METHOD PRIVATE ReferenceHMI
VAR_INPUT
END_VAR
Service_Handshake.AllocateMoveStructure 				REF= GVL_ADS.AllocateMoveStructure;
Service_Handshake.AllocateMoveStructure_Reverse 		REF= GVL_ADS.AllocateMoveStructure_Reverse;
Service_Handshake.EmptyRobotToTurnTableMove 			REF= GVL_ADS.EmptyRobotToTurnTableMove;
Service_Handshake.AllocateCircleMove 					REF= GVL_ADS.AllocateCircleMove;
Service_Handshake.TurnTableMove 						REF= GVL_ADS.TurnTableMove;
//Service_Handshake.AxesControl REF= GVL_ADS.AxesControl;
Service_Handshake.MachineReset 							REF= GVL_ADS.MachineReset;
Service_Handshake.RareFullBoxPush 						REF= GVL_ADS.RareFullBoxPush;
Service_Handshake.AutoMode_AllocateCircleMove 			REF= GVL_ADS.AutoMode_AllocateCircleMove;
Service_Handshake.AutoMode_RobotWarehouseMove 			REF= GVL_ADS.AutoMode_RobotWarehouseMove;
Service_Handshake.AutoMode_RobotAbsMove 				REF= GVL_ADS.AutoMode_RobotAbsMove;
Service_Handshake.AutoMode_EmptyBoxMove 				REF= GVL_ADS.AutoMode_EmptyBoxMove;
Service_Handshake.AutoMode_TurnTableMOve 				REF= GVL_ADS.AutoMode_TurnTableMOve;
Service_Handshake.AutoMode_AllocateMove 				REF= GVL_ADS.AutoMode_AllocateMove;
Service_Handshake.AutoMode_AllocateMove_Reverse 		REF= GVL_ADS.AutoMode_AllocateMove_Reverse;
Service_Handshake.AutoMode_AllocateBatchMode 			REF= GVL_ADS.AutoMode_AllocateBatchMode;
Service_Handshake.AutoMode_AllocateBatchMode_Reverse 	REF= GVL_ADS.AutoMode_AllocateBatchMode_Reverse;
Service_Handshake.AutoMode_SimpleAllocation_Batch 		REF= GVL_ADS.AutoMode_SimpleAllocation_Batch;
Service_Handshake.AutoMode_RareBoxMove 					REF= GVL_ADS.AutoMode_RareBoxMove;
Service_Handshake.AutoMode_OutBoxMove 					REF= GVL_ADS.AutoMode_OutBoxMove;
Service_Handshake.AutoMode_BoxMoveReverse 				REF= GVL_ADS.AutoMode_BoxMoveReverse;
Service_Handshake.AutoMode_WarehouseMove 				REF= GVL_ADS.AutoMode_WarehouseMove;
Service_Handshake.AutoMode_ErrorHandle 					REF= GVL_ADS.AutoMode_ErrorHandle;
Service_Handshake.AlarmAllocation 						REF= GVL_ADS.AlarmAllocation;
Service_Handshake.AutoMode_MoveConveyorJob 				REF= GVL_ADS.AutoMode_MoveConveyorJob;
Service_Handshake.AutoMode_WarehouseMotoWithRobotMove 	REF= GVL_ADS.AutoMode_WarehouseMotoWithRobotMove;
Service_Handshake.AutoMode_SimpleAllocate 				REF= GVL_ADS.AutoMode_SimpleAllocate;
Service_Handshake.AutoMode_PullOutConveyor 				REF= GVL_ADS.AutoMode_PullOutConveyor;
Service_Handshake.AutoMode_AddBoxes 					REF= GVL_ADS.AutoMode_AddBoxes;
Service_Handshake.MachineHome 							REF= GVL_ADS.MachineHome;
Service_Handshake.StorageRegionHome 					REF= GVL_ADS.StorageRegionHome;
Service_Handshake.AllocationRegionHome 					REF= GVL_ADS.AllocationRegionHome;
Service_Handshake.FGARegionHome 						REF= GVL_ADS.FGARegionHome;
Service_Handshake.StorageRegionMode 					REF= GVL_ADS.StorageRegionMode;
Service_Handshake.AllocationRegion 						REF= GVL_ADS.AllocationRegion;
Service_Handshake.FGARegionMode 						REF= GVL_ADS.FGARegionMode;
Service_Handshake.MachineMode 							REF= GVL_ADS.MachineMode;
Service_Handshake.OpPannel_Status 						REF= GVL_ADS.OpPannel_Status;
Service_Handshake.OpPannel_Ctrl 						REF= GVL_ADS.OpPannel_Ctrl;
Service_Handshake.FanucRobot_General 					REF= GVL_ADS.FanucRobot_General;
Service_Handshake.AutoMode_FeedInEmptyBoxWithRobot 		REF= GVL_ADS.AutoMode_FeedInEmptyBoxWithRobot;
Service_Handshake.AutoMode_ReloadRoundBeltBoxWithRobot 	REF= GVL_ADS.AutoMode_ReloadRoundBeltBoxWithRobot;
Service_Handshake.AutoMode_UpperFeedInConveyor 			REF= GVL_ADS.AutoMode_UpperFeedInConveyor;
//Service_Handshake.MachineState REF= GVL_ADS.MachineState;
Service_Handshake.AutoMode_RobotRegionMove_FeedInConveyor REF= GVL_ADS.AutoMode_RobotRegionMove_FeedInConveyor;
Service_Handshake.AutoMode_RobotRegionMove_AllocatedConveyor REF= GVL_ADS.AutoMode_RobotRegionMove_AllocatedConveyor;
Service_Handshake.AutoMode_RobotRegionMove_PullOutConveyor REF= GVL_ADS.AutoMode_RobotRegionMove_PullOutConveyor;
Service_Handshake.AutoMode_RobotRegionMove_BufferArea 	REF= GVL_ADS.AutoMode_RobotRegionMove_BufferArea;
Service_Handshake.AutoMode_RobotRegionMove_RoundBelt 	REF= GVL_ADS.AutoMode_RobotRegionMove_RoundBelt;
Service_Handshake.AutoMode_ShippingRobot_Left 			REF= GVL_ADS.AutoMode_ShippingRobot_Left;
Service_Handshake.AutoMode_ShippingRobot_Right 			REF= GVL_ADS.AutoMode_ShippingRobot_Right;
Service_Handshake.AutoMode_ShippingRobot_TransmitCVEnd 	REF= GVL_ADS.AutoMode_ShippingRobot_TransmitCVEnd;
Service_Handshake.AutoMode_SameSizeCVCamera 			REF= GVL_ADS.AutoMode_SameSizeCVCamera;
Service_Handshake.AutoMode_SameSizeCVCamera_Reverse 	REF= GVL_ADS.AutoMode_SameSizeCVCamera_Reverse;
Service_Handshake.AutoMode_DifferentCVCamera 			REF= GVL_ADS.AutoMode_DifferentCVCamera;

Service_Handshake.AllocationRobotNeedlingMove 			REF= GVL_ADS.AllocationRobotNeedlingMove;
Service_Handshake.RebootModbusDevices 					REF= GVL_ADS.RebootModbusDevices;
Service_Handshake.AutoMode_ShippingLeftSideTransCV 		REF= GVL_ADS.AutoMode_ShippingLeftSideTransCV;
Service_Handshake.AutoMode_ShippingRightSideTransCV 	REF= GVL_ADS.AutoMode_ShippingRightSideTransCV;
Service_Handshake.AutoMode_ShippingRobot_Buffer REF= GVL_ADS.AutoMode_ShippingRobot_Buffer;
Service_Handshake.AutoMode_ShippingRobot_PhotoStandByPos REF= GVL_ADS.AutoMode_ShippingRobot_PhotoStandByPos;
Service_Handshake.AutoMode_ShippingRobotTransfer REF= GVL_ADS.AutoMode_ShippingRobotTransfer;
Service_Handshake.AutoMode_ShippingPlateScan REF= GVL_ADS.AutoMode_ShippingPlateScan;

Service_Handshake.AutoMode_FeedInRoundBeltBoxToWareHouse REF= GVL_ADS.AutoMode_FeedInRoundBeltBoxToWareHouse;
Service_Handshake.AutoMode_WareHouseInnerPickToRoundBelt REF= GVL_ADS.AutoMode_WareHouseInnerPickToRoundBelt;
Service_Handshake.AutoMode_WareHouseInnerPickToRoundBeltBatch REF= GVL_ADS.AutoMode_WareHouseInnerPickToRoundBeltBatch;
Service_Handshake.AutoMode_FeedInRoundBeltBoxBatch REF= GVL_ADS.AutoMode_FeedInRoundBeltBoxBatch;

Service_Handshake.AutoMode_RobotSelfHoming REF= GVL_ADS.AutoMode_RobotSelfHoming;

Service_Handshake.AutoMode_ReverseBatchPick REF= GVL_ADS.AutoMode_ReverseBatchPick;
Service_Handshake.AutoMode_ReverseBoxToWareHouse REF= GVL_ADS.AutoMode_ReverseBoxToWareHouse;

Service_Handshake.BuzzCtrl REF= GVL_ADS.BuzzCtrl;
END_METHOD

METHOD RefShippingService
VAR_INPUT
END_VAR
ShippingService.AutoMode_ShippingRobot_Left 			REF= Service_Handshake.AutoMode_ShippingRobot_Left;
ShippingService.AutoMode_ShippingRobot_Right 			REF= Service_Handshake.AutoMode_ShippingRobot_Right;
ShippingService.AutoMode_ShippingRobot_TransmitCVEnd 	REF= Service_Handshake.AutoMode_ShippingRobot_TransmitCVEnd;
ShippingService.AutoMode_ShippingTransCV_LeftSide 		REF= Service_Handshake.AutoMode_ShippingLeftSideTransCV;
ShippingService.AutoMode_ShippingTransCV_RightSide 		REF= Service_Handshake.AutoMode_ShippingRightSideTransCV;
ShippingService.AutoMode_ShippingRobot_Buffer			REF= Service_Handshake.AutoMode_ShippingRobot_Buffer;
ShippingService.AutoMode_ShippingRobot_PhotoStandByPos  REF= Service_Handshake.AutoMode_ShippingRobot_PhotoStandByPos;
ShippingService.AutoMode_ShippingRobotTransfer			REF= Service_Handshake.AutoMode_ShippingRobotTransfer;
ShippingService.AutoMode_ShippingPlateScan				REF= Service_Handshake.AutoMode_ShippingPlateScan;
END_METHOD

METHOD PRIVATE RefStorageService
VAR_INPUT
END_VAR
StorageService.AutoMode_ReloadRoundBeltBoxWithRobot	REF= Service_Handshake.AutoMode_ReloadRoundBeltBoxWithRobot;
StorageService.AutoMode_FeedInEmptyBoxWithRobot REF= Service_Handshake.AutoMode_FeedInEmptyBoxWithRobot;
StorageService.AutoMode_RobotRegionMove_FeedInConveyor REF= Service_Handshake.AutoMode_RobotRegionMove_FeedInConveyor;
StorageService.AutoMode_RobotRegionMove_AllocatedConveyor REF= Service_Handshake.AutoMode_RobotRegionMove_AllocatedConveyor;
StorageService.AutoMode_RobotRegionMove_PullOutConveyor REF= Service_Handshake.AutoMode_RobotRegionMove_PullOutConveyor;
StorageService.AutoMode_RobotRegionMove_BufferArea REF= Service_Handshake.AutoMode_RobotRegionMove_BufferArea;
StorageService.AutoMode_RobotRegionMove_RoundBelt REF= Service_Handshake.AutoMode_RobotRegionMove_RoundBelt;
StorageService.AutoMode_UpperFeedInConveyor REF=  Service_Handshake.AutoMode_UpperFeedInConveyor;
StorageService.AutoMode_AddBoxes REF= Service_Handshake.AutoMode_AddBoxes;
StorageService.AutoMode_PullOutConveyor REF= Service_Handshake.AutoMode_PullOutConveyor;
StorageService.AutoMode_RobotAbsMove REF=  Service_Handshake.AutoMode_RobotAbsMove;
StorageService.AutoMode_WarehouseMotoWithRobotMove REF= Service_Handshake.AutoMode_WarehouseMotoWithRobotMove;
StorageService.RebootModbusDevices REF= Service_Handshake.RebootModbusDevices;
StorageService.AutoMode_FeedInRoundBeltBoxToWareHouse REF= Service_Handshake.AutoMode_FeedInRoundBeltBoxToWareHouse;
StorageService.AutoMode_WareHouseInnerPickToRoundBelt REF= Service_Handshake.AutoMode_WareHouseInnerPickToRoundBelt;
StorageService.AutoMode_WareHouseInnerPickToRoundBeltBatch REF= Service_Handshake.AutoMode_WareHouseInnerPickToRoundBeltBatch;
StorageService.AutoMode_FeedInRoundBeltBoxBatch REF= Service_Handshake.AutoMode_FeedInRoundBeltBoxBatch;
StorageService.AutoMode_RobotSelfHoming REF= Service_Handshake.AutoMode_RobotSelfHoming;
END_METHOD

END_FUNCTION_BLOCK

// ---- Library/00_PackML/01_ObjectBase/FB_ModeBase_V2.TcPOU
{attribute 'reflection'}
FUNCTION_BLOCK FB_ModeBase_V2 IMPLEMENTS I_UnitState, I_ErrorElement
VAR_INPUT
    eModeCommand  : E_UnitMode; // Mode from superior Unit
    eStateCommand : E_PMLCommand := ePMLCommand_Abort; // Command fro a new state from supterior unit
    PackTag       : REFERENCE TO ST_PackMLv30; // 
END_VAR
VAR_OUTPUT
    eModeCurrent  : E_UnitMode;
    eStateCurrent : E_PMLState;
END_VAR
VAR
    {attribute 'instance-path'}
    {attribute 'noinit'}
    _strName : STRING(255); // Instance path of the FB for Diagnostic

    fbUnitModeManager : PML_UnitModeManager; //The PML_UnitModeManager manage the Modechanges
    fbStateMachine    : PML_StateMachine; //The PML_StateMachine mangae the Statechanges

    eModeChange     : eModeChangeState; // This value is used to control mode change flow
    AllowModeChange : BOOL;
    nLastState      : E_PMLState; //Variable to store last state
    xError           : BOOL;
    xErrorID         : DINT;
    xErrorMsg        : T_MaxString;
	iErrorCount : INT;
	arAlarmTrigPtr : ARRAY[1..Tc3_PackML_V2.MaxAlarms] OF POINTER TO BOOL;
	arAlarmMsg : ARRAY[1..Tc3_PackML_V2.MaxAlarms] OF POINTER TO STRING;
	iErrorReflashIndex : INT;
END_VAR

CASE eModeChange OF
    eModeChangeState.WaitingRequest:
        // check unit is in the stand still, allow to change mode
        AllowModeChange := M_ModeChangeCheck();

        IF AllowModeChange AND (eModeCommand <> eModeCurrent) THEN
            eModeChange := eModeChangeState.StartingUnitModeManager;
        END_IF
    eModeChangeState.StartingUnitModeManager:
        fbUnitModeManager.bExecute             := TRUE;
        PackTag.Status.UnitModeChangeInProcess := TRUE;

        IF fbUnitModeManager.bDone THEN
            fbUnitModeManager.bExecute             := FALSE;
            eModeChange                            := eModeChangeState.WaitingRequest;
            PackTag.Status.UnitModeChangeInProcess := FALSE;
        ELSIF fbUnitModeManager.bError THEN
            fbUnitModeManager.bExecute := FALSE;
            nLastState                 := PackTag.Status.StateCurrent;
            eModeChange                := eModeChangeState.ErrorHandling;
        END_IF
    eModeChangeState.ErrorHandling:
        //ErrorHanddling
		eModeChange := 0; 
//        IF PackTag.Command.UnitModeChangeRequest THEN
//            eModeChange := 0;
//        ELSIF nLastState <> PackTag.Status.StateCurrent THEN
//            ;
//        END_IF
END_CASE

fbUnitModeManager(bExecute :=,
                  eModeCommand := eModeCommand,
                  eState := eStateCurrent,
                  eModeStatus => eModeCurrent,
                  sModeStatus =>,
                  bDone =>,
                  bError =>,
                  nErrorId =>);

IF fbUnitModeManager.eModeStatus <> E_UnitMode.Undefined THEN
    fbStateMachine(eMode := eModeCommand,
                   eCommand := eStateCommand,
                   stSubUnitInfoRef :=,
                   stOptions :=,
                   eState => eStateCurrent,
                   sState =>,
                   bError =>,
                   nErrorID =>);
END_IF

//One of the methods is executing  by the actual state
CASE eStateCurrent OF
    ePMLState_Undefined:
        M_Undefined();
    ePMLState_Clearing:
        M_Clearing();
    ePMLState_Stopped:
        M_Stopped();
    ePMLState_Starting:
        M_Starting();
    ePMLState_Idle:
        M_Idle();
    ePMLState_Suspended:
        M_Suspended();
    ePMLState_Execute:
        M_Execute();
    ePMLState_Stopping:
        M_Stopping();
    ePMLState_Aborting:
        M_Aborting();
    ePMLState_Aborted:
        M_Aborted();
    ePMLState_Holding:
        M_Holding();
    ePMLState_Held:
        M_Held();
    ePMLState_Unholding:
        M_Unholding();
    ePMLState_Suspending:
        M_Suspending();
    ePMLState_Unsuspending:
        M_Unsuspending();
    ePMLState_Resetting:
        M_Resetting();
    ePMLState_Completing:
        M_Completing();
    ePMLState_Complete:
        M_Complete();
END_CASE

Act_ErrorSync();

ACTION Act_ErrorSync:
FOR iErrorReflashIndex := 1 TO MaxAlarms DO
    IF arAlarmTrigPtr[iErrorReflashIndex] <> 0 THEN
        PackTag.Admin.Alarm[iErrorReflashIndex].Trigger := arAlarmTrigPtr[iErrorReflashIndex]^;
		//PackTag.Admin.Alarm[iErrorReflashIndex].Message := arAlarmMsg[iErrorReflashIndex]^;
    END_IF
END_FOR
END_ACTION

METHOD M_Aborted
M_StateComplete();
END_METHOD

METHOD M_Aborting
M_StateComplete();
END_METHOD

METHOD M_Clearing
M_StateComplete();
END_METHOD

METHOD M_Complete
M_StateComplete();
END_METHOD

METHOD M_Completing
M_StateComplete();
END_METHOD

METHOD M_Execute
M_StateComplete();
END_METHOD

METHOD M_GetError
VAR_INPUT
END_VAR
VAR_OUTPUT
	Error : BOOL;
	ErrorID : DINT;
	ErrorMsg : T_MaxString;
END_VAR
Error := xError;
ErrorID := xErrorID;
ErrorMsg := xErrorMsg;
END_METHOD

METHOD PUBLIC M_GetName :STRING
VAR_INPUT
END_VAR
M_GetName := _strName;
END_METHOD

METHOD M_Held
M_StateComplete();
END_METHOD

METHOD M_Holding
M_StateComplete();
END_METHOD

METHOD M_Idle
M_StateComplete();
END_METHOD

METHOD M_ModeChageAutoCheck : BOOL
VAR_INPUT
END_VAR
CASE eStateCurrent OF
	ePMLState_Aborted,ePMLState_Stopped,ePMLState_Idle :
		// Allow unit change mode to Auto
		M_ModeChageAutoCheck := TRUE;
	ePMLState_Undefined:
		M_ModeChageAutoCheck := TRUE;
END_CASE
END_METHOD

METHOD M_ModeChangeCheck : BOOL
VAR_INPUT
END_VAR
VAR_INST
    ManualAllowChange : BOOL;
    AutoAllowChange   : BOOL;
    HomingAllowChange : BOOL;
	MantainaceAllowChange : BOOL;
END_VAR
ManualAllowChange     := M_ModeChangeManualCheck();
AutoAllowChange       := M_ModeChageAutoCheck();
HomingAllowChange     := M_ModeChangeHomingCheck();
MantainaceAllowChange := M_ModeChangeMantainaceCheck();

M_ModeChangeCheck := ManualAllowChange AND AutoAllowChange AND HomingAllowChange AND MantainaceAllowChange;
END_METHOD

METHOD M_ModeChangeHomingCheck : BOOL
VAR_INPUT
END_VAR
CASE eStateCurrent OF
	ePMLState_Aborted,ePMLState_Stopped,ePMLState_Idle :
		// Allow unit change mode to Homing
		M_ModeChangeHomingCheck := TRUE;
	ePMLState_Undefined:
		M_ModeChangeHomingCheck := TRUE;

END_CASE
END_METHOD

METHOD M_ModeChangeMantainaceCheck : BOOL
VAR_INPUT
END_VAR
CASE eStateCurrent OF
	ePMLState_Aborted,ePMLState_Stopped,ePMLState_Idle :
		// Allow unit change mode to Mantainace
		M_ModeChangeMantainaceCheck := TRUE;
	ePMLState_Undefined:
		M_ModeChangeMantainaceCheck := TRUE;

END_CASE
END_METHOD

METHOD M_ModeChangeManualCheck : BOOL
VAR_INPUT
END_VAR
CASE eStateCurrent OF
	ePMLState_Aborted,ePMLState_Stopped,ePMLState_Idle :
		// Allow unit change mode to Manual
		M_ModeChangeManualCheck := TRUE;
	ePMLState_Undefined:
		M_ModeChangeManualCheck := TRUE;

END_CASE
END_METHOD

METHOD M_Resetting
M_StateComplete();
END_METHOD

METHOD M_Starting
M_StateComplete();
END_METHOD

METHOD M_StateComplete
//the actual state is completed
fbStateMachine.M_StateComplete();
END_METHOD

METHOD M_Stopped
M_StateComplete();
END_METHOD

METHOD M_Stopping
M_StateComplete();
END_METHOD

METHOD M_Suspended
M_StateComplete();
END_METHOD

METHOD M_Suspending
M_StateComplete();
END_METHOD

METHOD M_Undefined
M_StateComplete();
END_METHOD

METHOD M_Unholding
M_StateComplete();
END_METHOD

METHOD M_Unsuspending
M_StateComplete();
END_METHOD

METHOD RegisterAlarm
VAR_INPUT
    Trigger  : REFERENCE TO BOOL;
    ID       : DINT;
    value    : DINT;
    Message  : STRING;
    Category : DINT;
END_VAR
VAR_INST
    iLoopIndex : INT;
    HasSameID  : BOOL := FALSE;
    FoundIndex : INT := 0;
    FoundCount : INT := 0;
END_VAR
// VAR_INST 必須在每次呼叫開頭重置，否則一旦某次找到重複就會卡 TRUE，
// 後面新 ID 都會被當成已存在而拒絕註冊（iErrorCount 不再增加）。
HasSameID := FALSE;
FoundIndex := 0;
FoundCount := 0;

FOR iLoopIndex := 1 TO MaxAlarms DO
    IF PackTag.Admin.Alarm[iLoopIndex].ID = ID THEN
        IF NOT HasSameID THEN
            HasSameID := TRUE;
            FoundIndex := iLoopIndex;

			EXIT;
        END_IF
		PackTag.Admin.Alarm[iLoopIndex].Message := Message;
        FoundCount := FoundCount + 1;
    END_IF
END_FOR

//IF NOT HasSameID THEN
//    PackTag.Admin.Alarm[iErrorCount+1].ID := ID;
//    PackTag.Admin.Alarm[iErrorCount+1].Value := value;
//    PackTag.Admin.Alarm[iErrorCount+1].Message := Message;
//    PackTag.Admin.Alarm[iErrorCount+1].Category := Category;
//	arAlarmTrigPtr[iErrorCount+1] := ADR(Trigger);
//	//arAlarmMsg[iErrorCount+1] := ADR(Message);
//	iErrorCount := iErrorCount +1 ;
//END_IF

IF NOT HasSameID THEN
    PackTag.Admin.Alarm[iErrorCount + 1].ID       := ID;
    PackTag.Admin.Alarm[iErrorCount + 1].Value    := value;
    PackTag.Admin.Alarm[iErrorCount + 1].Message  := Message;
    PackTag.Admin.Alarm[iErrorCount + 1].Category := Category;
    arAlarmTrigPtr[iErrorCount + 1]               := ADR(Trigger);
    iErrorCount                                   := iErrorCount + 1;
ELSE
    // 找到既有 Alarm ID 時，也要回寫最新訊息，
    // 避免初始化時的空字串一路保留到 ADS 顯示端。
    PackTag.Admin.Alarm[FoundIndex].Value    := value;
    PackTag.Admin.Alarm[FoundIndex].Message  := Message;
    PackTag.Admin.Alarm[FoundIndex].Category := Category;
END_IF
END_METHOD

END_FUNCTION_BLOCK

// ---- Library/10_Machine/18_HMI_Handshake/FB_HmiHandShake.TcPOU
FUNCTION_BLOCK FB_HmiHandShake EXTENDS BATW_Base.FB_ActionBasic
VAR_INPUT
    xEnable        : BOOL;
    CylinderStatus : ST_CylinderStatus;
    MotorStatus    : ST_MotorStatus;
    AxesStatus     : ST_AXES_STATUS;
	FanucRobot : REFERENCE TO UNI_FanucRobotList;
END_VAR
VAR_OUTPUT
	//AllocatingManual : st_ads_AllocateMoveStructure;
END_VAR
VAR
    StateBehaviour : CBML.LConC;
	//HMI_Handshake_Old : REFERENCE TO ST_HMI_Handshake;
END_VAR

THIS^.IBehaviourModel := StateBehaviour;
StateBehaviour(xEnable := xEnable, xBusy => xBusy, xError => xError);

METHOD CleanupAction
VAR_INPUT
    xAbortProposed   : BOOL;
    iErrorIDProposed : INT;
END_VAR
VAR_OUTPUT
    xComplete : BOOL := TRUE;
    xAbort    : BOOL := xAbortProposed;
    iErrorID  : INT := iErrorIDProposed;
END_VAR
END_METHOD

METHOD CyclicAction
VAR_INPUT
    itfTimingController : CBML.ITimingController;
END_VAR
VAR_OUTPUT
    xComplete : BOOL := TRUE;
    iErrorID  : INT := 0;
END_VAR
GetIOStatus();
GetAxesStatus();
GetMotorStatus();
GetCylinderStatus();
SetMachineParemeter();
//AllocatingManual := GVL_ADS.AllocateMoveStructure;
FanucRobot.List.StorageRobot.VelocityCommand := LREAL_TO_INT( GVL_HMI.Setup.StorageRobot.RobotVelocity);
FanucRobot.List.ShippingRobot.VelocityCommand := LREAL_TO_INT( GVL_HMI.Setup.ShippingRobot.RobotVelocity);
END_METHOD

METHOD ExitAction
VAR_INPUT
    xAfterCleanup : BOOL;
    xInCopyCode   : BOOL;
END_VAR
END_METHOD

(* This method is used to read DAS servo status and send to GVL_HMI
*)
METHOD PRIVATE GetAxesStatus
VAR_INPUT
END_VAR
// Read Axes status
GVL_HMI.Status.Axes.Allocate_X := M_GetAxisStatus(AxisNo.Allocate_X);
GVL_HMI.Status.Axes.Allocate_Y := M_GetAxisStatus(AxisNo.Allocate_Y);
GVL_HMI.Status.Axes.OutRobot_X := M_GetAxisStatus(AxisNo.OutRobot_X);
GVL_HMI.Status.Axes.OutRobot_Y := M_GetAxisStatus(AxisNo.OutRobot_Y);
GVL_HMI.Status.Axes.RoundBelt := M_GetAxisStatus(AxisNo.RoundBelt);
GVL_HMI.Status.Axes.TurnTable := M_GetAxisStatus(AxisNo.TurnTable);
GVL_HMI.Status.Axes.RackMotor := M_GetAxisStatus(AxisNo.RackMotor);
END_METHOD

METHOD PRIVATE GetCylinderStatus
VAR_INPUT
END_VAR
GVL_HMI.Status.Cylinders := CylinderStatus;
END_METHOD

METHOD PRIVATE GetIOStatus
VAR_INPUT
END_VAR
// Read  PLC Input Signal
GVL_HMI.IOMonitor.Input.X0  := GVL_Input.uniDI.stDIList.X0;
GVL_HMI.IOMonitor.Input.X1  := GVL_Input.uniDI.stDIList.X1;
GVL_HMI.IOMonitor.Input.X2  := GVL_Input.uniDI.stDIList.X2;
GVL_HMI.IOMonitor.Input.X3  := GVL_Input.uniDI.stDIList.X3;
GVL_HMI.IOMonitor.Input.X4  := GVL_Input.uniDI.stDIList.X4;
//GVL_HMI.IOMonitor.Input.X5  := GVL_Input.uniDI.stDIList.X0;
GVL_HMI.IOMonitor.Input.X6  := GVL_Input.uniDI.stDIList.X6;
GVL_HMI.IOMonitor.Input.X7  := GVL_Input.uniDI.stDIList.X7;
GVL_HMI.IOMonitor.Input.X8  := GVL_Input.uniDI.stDIList.X8;
GVL_HMI.IOMonitor.Input.X9  := GVL_Input.uniDI.stDIList.X9;
GVL_HMI.IOMonitor.Input.X10  := GVL_Input.uniDI.stDIList.X10;
GVL_HMI.IOMonitor.Input.X11  := GVL_Input.uniDI.stDIList.X11;
// Read PLC Output signal
GVL_HMI.IOMonitor.Output := GVL_Output.uniDO.stDIList;
// Read Wheelhous ModbusRTU sensor signal
//GVL_HMI.IOMonitor.Input.arWheelhouseInput := ComModbusRTU.arr485sensor;

//RS485 Jidian Version edited Gamin 20251120
GVL_HMI.IOMonitor.Input.arWheelhouseInput := MAIN2_RS485.arr485sensor;
END_METHOD

METHOD PRIVATE GetMotorStatus
VAR_INPUT
END_VAR
GVL_HMI.Status.Motor := MotorStatus;
END_METHOD

(* This method is used to read single axis status accroding AxisNo
*)
METHOD M_GetAxisStatus : ST_SINGLEAXIS_STATUS
VAR_INPUT
	AxisNo : AxisNo;
END_VAR
M_GetAxisStatus.ActPos := arAxisCtrl_gb[AxisNo].Admin.Axis.NcToPlc.ActPos;
M_GetAxisStatus.ActVel := arAxisCtrl_gb[AxisNo].Admin.Axis.NcToPlc.ActVelo;
M_GetAxisStatus.Error := arAxisCtrl_gb[AxisNo].Admin.Axis.Status.Error;
IF AxisNo = 4 THEN
	M_GetAxisStatus.Homed := GVL_Machine.AllocatYAxisHome;
ELSE
	M_GetAxisStatus.Homed := arAxisCtrl_gb[AxisNo].Admin.Axis.Status.Homed;
END_IF

M_GetAxisStatus.CmdDone := arAxisStatus_gb[AxisNo].Admin.CmdDone;
M_GetAxisStatus.DriveTemp := 400;
M_GetAxisStatus.MotorTemp := 600;
END_METHOD

METHOD ResetAction
VAR_OUTPUT
    xComplete : BOOL := TRUE;
END_VAR
END_METHOD

METHOD PRIVATE SetMachineParemeter
VAR_INPUT
END_VAR
GVL_Machine.RemoteData := GVL_HMI.Setup;
END_METHOD

METHOD StartAction
VAR_OUTPUT
    xComplete : BOOL := TRUE;
    iErrorID  : INT := 0;
END_VAR
END_METHOD

END_FUNCTION_BLOCK

// ---- Library/20_MachineUnits/22_AllocateArea/FB_AllocateAreaWithRoundbelt.TcPOU
FUNCTION_BLOCK FB_AllocateAreaWithRoundbelt EXTENDS FB_ModeBase_V2 IMPLEMENTS I_UnitState
VAR_INPUT
    INPUT       : REFERENCE TO ST_InputTable;
    OUTPUT      : REFERENCE TO ST_OutputTable;
    CurrentData : ST_SetupPara;
    // Componets
    Cylinder 	: REFERENCE TO UNI_CylinderList;
    Service  	: REFERENCE TO ST_AllocateService;
    Motor    	: REFERENCE TO UNI_MotorList;
    SameSizeCVRequest : REFERENCE TO ST_SameSizeCVRequest;	// Phase 2 仲裁,傳到 fbReverseBatchPickAndPhoto / fbReverseBoxToWareHouse / fbSameSizeCVCamera_Reverse
    Reset       : REFERENCE TO BOOL;
	Stop 		: REFERENCE TO BOOL;
	bStopMem 	: REFERENCE TO BOOL;
END_VAR
VAR_OUTPUT
	Homed : BOOL;
END_VAR
VAR
	Abort	: BOOL;

	// 連動暫停 - 任一 Service 錯誤時暫停所有其他 Service
	_bAnyServiceError : BOOL;

    InitDone          : BOOL;
    Clip              : U_Cylinders;
    Cylinders         : U_Cylinders;
    OutRobotCylinders : Uni_DuoCylinders;
    OutRobotClips     : Uni_DuoCylinders;

    i : INT;
    //============== Service====================
    // Allocate Home
    fbAllocateHome : FB_AllocateAreaHome;
    //RoundBelt
    RoundBeltControl  : FB_RoundBeltService;
    _RoundBeltMoveJob : st_AllocateCircleMoveStructure;
    //RoundBeltMoveJob_Internal 	: st_AllocateCircleMoveStructure;		
    RoundBeltControlAccess               : E_RoundBeltControlAccess := E_RoundBeltControlAccess.Host;
    RoundBeltMoveJob_Ctrl                : ST_CommandBasic;
    RoundBeltMoveJob_Ctrl_Batch          : ST_CommandBasic;
    RoundBeltMoveJob_Status              : ST_StatusBasic;
    RoundBeltMoveJob_Position            : LREAL;
    RoundBeltMoveJob_Position_FanucRobot : LREAL;
    //TurnTable
    TurnTableControl : FB_TurnTableService;

    //Allocating
    fb_AllocateBatchMode        : FB_AllocateMoveAutoBatchMode;
    AutoAllocateJobBatch_Ctrl   : st_AllocateMoveAutoBatchMode_Ctrl;
    AutoAllocateJobBatch_Status : st_AllocateMoveAutoBatchMode_Status;
    bAutoAllocateJobDryRun      : BOOL;

	  //Allocating reverse
    fb_AllocateBatchMode_Reverse        : FB_AllocateMoveAutoBatchMode_Reverse;
    AutoAllocateJobBatch_Reverse_Ctrl   : st_AllocateMoveAutoBatchMode_Ctrl;
    AutoAllocateJobBatch_Reverse_Status : st_AllocateMoveAutoBatchMode_Status;
   
	
    //OutRobot EmptyBoxMove
    fbOutRobot_EmptyBoxMove        : FB_OutRobot_EmptyBoxMove;
    fbOutRobot_EmptyBoxMove_Ctrl   : ST_CommandBasic;
    fbOutRobot_EmptyBoxMove_Status : ST_StatusBasic;

    //OutRobot RareBoxMove
    fbOutRobot_RareBoxMove        : FB_OutRobot_RareBoxMove;
    fbOutRobot_RareBoxMove_Ctrl   : ST_CommandBasic;
    fbOutRobot_RareBoxMove_Status : ST_StatusBasic;

    //OutRobot BoxMoveReverse	
    fbOutRobot_BoxMoveReverse        : FB_OutRobot_BoxMoveReverse;
    fbOutRobot_BoxMoveReverse_Ctrl   : ST_CommandBasic;
    fbOutRobot_BoxMoveReverse_Status : ST_StatusBasic;

	//OutRobot TurnTable to RoundBelt
	fbOutRobot_TurnTableToRoundBelt: FB_OutRobot_BoxMoveTurnTableToRoundBelt;
	fbOutRobot_TurnTableToRoundBel_Ctrl   : ST_CommandBasic;
    fbOutRobot_TurnTableToRoundBel_Status : ST_StatusBasic;
	
    //TransCV Camera
    fbSameSizeCVCamera  		: FB_SameSizeCVCamera;
	fbSameSizeCVCamera_Reverse 	: FB_SameSizeCVCamera_Reverse;
    fbDifferentCVCamera 		: FB_DifferentCVCamera;
	// 逆向拍照批次入料
	fbReverseBatchPickAndPhoto 	: FB_SameSizeCV_ReverseBatchPickAndPhoto;
	fbReverseBoxToWareHouse    	: FB_SameSizeCV_ReverseBoxToWareHouse;
	TransCV_Press 				: BOOL :=FALSE;

    // Round belt
    AutoRotatebelt_Internal_Ctrl   : st_RoundBeltAutoSingleMove_Ctrl;
    AutoRotatebelt_Internal_Status : st_RoundBeltAutoSingleMove_Status;
    _AutoRotatebelt_Ctrl           : st_RoundBeltAutoSingleMove_Ctrl;
    _AutoRotatebelt_Status         : st_RoundBeltAutoSingleMove_Status;
    bInternalRotateBeltRequest     : BOOL;
    bReloadRotateBeltRequest       : BOOL;

    // Pullout

    fbPulloutCV                 : FB_PullOutConveyorAction;
    _AutoPullout_Ctrl           : ST_AutoPullOutConveyorCommand;
    _AutoPullout_Status         : ST_AutoPullOutConveyorSatus;
    _AutoPullout_Info           : ST_PullOutConveyorInfo;
    AutoPullout_Internal_Ctrl   : ST_AutoPullOutConveyorCommand;
    AutoPullout_Internal_Status : ST_AutoPullOutConveyorSatus;
    AutoPullout_Internal_Info   : ST_PullOutConveyorInfo;
    RobotPullout_Internal_Ctrl   : ST_AutoPullOutConveyorCommand;
    RobotPullout_Internal_Status : ST_AutoPullOutConveyorSatus;
    RobotPullout_Internal_Info   : ST_PullOutConveyorInfo;
	fbPulloutCV_BTNCtrl			:FB_PullOutConveyorBtnCtrl;

    PulloutControlAccess        : E_RoundBeltControlAccess := E_RoundBeltControlAccess.Host;
    bPulloutConveyorInternCtrl  : BOOL;
	
	// TurnTable
	 _TurnTableMove                      :  st_ads_OneAxisMoveWithPosition;
	 
	 //AllocateRobotNeedlingMove
	 fbAllocateRobotNeedlingMove		: FB_AllocateRobotNeedlingMove;

END_VAR

SUPER^();
IF __ISVALIDREF(PackTag)  THEN
	
    eModeCommand  := PackTag.Command.UnitMode;
    eStateCommand := PackTag.Command.CntrlCmd;
ELSE
    RETURN;
END_IF

IF __ISVALIDREF(Cylinder) THEN
	
	Clip.stCylinders.Cylinder0 REF= Cylinder.List.fbAllocateRobot_LeftClamp1;
	Clip.stCylinders.Cylinder1 REF= Cylinder.List.fbAllocateRobot_LeftClamp2;
	Clip.stCylinders.Cylinder2 REF= Cylinder.List.fbAllocateRobot_RightClamp1;
	Clip.stCylinders.Cylinder3 REF= Cylinder.List.fbAllocateRobot_RightClamp2;
	Cylinders.stCylinders.Cylinder0 REF= Cylinder.List.fbAllocateRobot_LeftVert1;
	Cylinders.stCylinders.Cylinder1 REF= Cylinder.List.fbAllocateRobot_LeftVert2;
	Cylinders.stCylinders.Cylinder2 REF= Cylinder.List.fbAllocateRobot_RightVert1;
	Cylinders.stCylinders.Cylinder3 REF= Cylinder.List.fbAllocateRobot_RightVert2;
	
	OutRobotCylinders.stCylinders.Cylinder1 REF= Cylinder.List.fbOutRobot_AsideVert;
	OutRobotCylinders.stCylinders.Cylinder2 REF= Cylinder.List.fbOutRobot_BsideVert;
	OutRobotClips.stCylinders.Cylinder1 REF= Cylinder.List.fbOutRobot_AsideClamp;
	OutRobotClips.stCylinders.Cylinder2 REF= Cylinder.List.fbOutRobot_BsideClamp;
	
END_IF

ACTION A00_Service:
// ============================================================================
// 連動暫停邏輯 - 任一 Service 錯誤時，暫停所有其他 Service
// ============================================================================
_bAnyServiceError := FALSE;
//	_RoundBeltMoveJob.HandShake.Error OR
//	_TurnTableMove.HandShake.Error OR
//	AutoAllocateJobBatch_Status.bError OR
//	AutoAllocateJobBatch_Reverse_Status.bError OR
//	Service.AutoMode_EmptyBoxMove.HandShake.Error OR
//	Service.AutoMode_RareBoxMove.HandShake.Error OR
//	Service.AutoMode_BoxMoveReverse.HandShake.Error OR
//	Service.AutoMode_DifferentCVCamera.Status.Error OR
//	fbOutRobot_TurnTableToRoundBel_Status.Error OR
//	Service.AutoMode_SameSizeCVCamera.Status.Error OR
//	_AutoPullout_Status.Error OR
//	Service.AllocateRobotNeedlingMove.Status.Error;

fbAllocateHome(
	xDone=> ,
	xBusy=> ,
	xError=> ,
	xExecute:= ,
	xAbort:= THIS^.Abort OR _bAnyServiceError,
	Homed := Homed,
	Cylinder:= Cylinder, 
	Motor:= Motor, 
	CurrentData:= CurrentData, 
	TimeOut:= , 
	xAborted=> , 
	iErrorID=> , 
	ErrorMsg=> ,
	AxisHomingRequest =>);
	//Service.AllocateRegionHome.Homed:= bHomed;

RoundBeltControl(
	xDone=> _RoundBeltMoveJob.HandShake.Done,
	xBusy=> _RoundBeltMoveJob.HandShake.Busy,
	xError=> _RoundBeltMoveJob.HandShake.Error,
	xExecute:= _RoundBeltMoveJob.HandShake.Execute,
	xAbort:= THIS^.Abort OR _bAnyServiceError,
	TargetStation:= LREAL_TO_INT( _RoundBeltMoveJob.Position),
	Cylinder:= Cylinder, 
	TimeOut:= , 
	xAborted=> , 
	iErrorID=> , 
	ErrorMsg=> ,
	AxisRoundMoveRequest => ,
	Pause	:= bStopMem);
	
TurnTableControl(
	xDone=> _TurnTableMove.HandShake.Done,
	xBusy=> _TurnTableMove.HandShake.Busy,
	xError=> _TurnTableMove.HandShake.Error,
	xExecute:= _TurnTableMove.HandShake.Execute,
	xAbort:= THIS^.Abort OR _bAnyServiceError,
	iTurnTableTarget:= LREAL_TO_INT(_TurnTableMove.Position),
	Cylinder:= Cylinder, 
	//TimeOut:= , 
	xAborted=> , 
	iErrorID=> , 
	ErrorMsg=> ,
	bTurnTableMoveRequest=>,
	Pause := bStopMem);
	
fb_AllocateBatchMode(
	Execute:= AutoAllocateJobBatch_Ctrl.bExecute,
	Abort:= THIS^.Abort OR _bAnyServiceError,
	Reset:= AutoAllocateJobBatch_Ctrl.bReset,
	ObjectName:= 'Allocate One process',
	Busy=> AutoAllocateJobBatch_Status.bBusy,
	Done=> AutoAllocateJobBatch_Status.bDone,
	Aborted=> ,
	Error=> AutoAllocateJobBatch_Status.bError,
	ErrorID=>AutoAllocateJobBatch_Status.ErrorID ,
	Status=>AutoAllocateJobBatch_Status.Status ,
	UniqueErrorCode=> , 
	SimpleAllocateMode:= AutoAllocateJobBatch_Ctrl.bSimpleAllocation, 
	bOccupied:=AutoAllocateJobBatch_Ctrl.bOccupied, 
	Clips:= Clip.Cylinders, 
	cylinders:= Cylinders.Cylinders, 
	TurnTable_Press:= Cylinder.List.fbTurntable_Press, 
	RoundBelt_Press:= Cylinder.List.fbRoundBelt_WorkZone_Press, 
	AutoAllocateJobBatch_Ctrl:= AutoAllocateJobBatch_Ctrl, 
	INPUT:= INPUT, 
	OUTPUT:= OUTPUT, 
	NrOfAllocateCylinder:= 4, 
	CurrentData:= CurrentData, 
	bAutoAllocateJobDryRun:= bAutoAllocateJobDryRun, // Dry run : No round belt move
	ProcessedIndex=> AutoAllocateJobBatch_Status.iIndex,
	RoundBeltMoveJob_Ctrl =>,
	RoundBeltMoveJob_Status := RoundBeltMoveJob_Status,
	RoundBeltMoveJob_Position =>	 ,
	Pause := bStopMem);
	
	IF fb_AllocateBatchMode.SimpleAllocateMode THEN
		 Service.AutoMode_SimpleAllocation_Batch.WorkedID:= AutoAllocateJobBatch_Status.iIndex;
	ELSE
		 Service.AutoMode_AllocateBatchMode.WorkedID:= AutoAllocateJobBatch_Status.iIndex;
	END_IF
fb_AllocateBatchMode_Reverse(
	Execute:=AutoAllocateJobBatch_Reverse_Ctrl.bExecute ,
	Abort:= THIS^.Abort OR _bAnyServiceError,
	Reset:= AutoAllocateJobBatch_Reverse_Ctrl.bReset,
	Pause:= bStopMem,
	ObjectName:= 'Allocate batch reverse',
	Busy=> AutoAllocateJobBatch_Reverse_Status.bBusy,
	Done=> AutoAllocateJobBatch_Reverse_Status.bDone,
	Aborted=> AutoAllocateJobBatch_Reverse_Status.bAborted,
	Error=> AutoAllocateJobBatch_Reverse_Status.bError,
	ErrorID=> AutoAllocateJobBatch_Reverse_Status.ErrorID,
	Status=> AutoAllocateJobBatch_Reverse_Status.Status,
	UniqueErrorCode=> ,  
	bOccupied:= AutoAllocateJobBatch_Reverse_Ctrl.bOccupied, 
	Clips:= Clip.Cylinders, 
	cylinders:= Cylinders.Cylinders, 
	TurnTable_Press:= Cylinder.List.fbTurntable_Press, 
	RoundBelt_Press:= Cylinder.List.fbRoundBelt_WorkZone_Press, 
	AutoAllocateJobBatch_Reverse_Ctrl:= AutoAllocateJobBatch_Reverse_Ctrl, 
	INPUT:= INPUT, 
	OUTPUT:= OUTPUT, 
	NrOfAllocateCylinder:=4 , 
	CurrentData:= CurrentData, 
	bAutoAllocateJobDryRun:= bAutoAllocateJobDryRun, 
	RoundBeltMoveJob_Ctrl=> , 
	ProcessedIndex=> AutoAllocateJobBatch_Reverse_Status.iIndex,
	RoundBeltMoveJob_Status := RoundBeltMoveJob_Status,
	RoundBeltMoveJob_Position =>);

	
fbOutRobot_EmptyBoxMove(
	Execute:= Service.AutoMode_EmptyBoxMove.HandShake.Execute,
	Abort:= THIS^.Abort OR _bAnyServiceError,
	Reset:= Reset ,
	ObjectName:= 'fbOutRobot_EmptyBoxMove', 
	Busy=> Service.AutoMode_EmptyBoxMove.HandShake.Busy, 
	Done=> Service.AutoMode_EmptyBoxMove.HandShake.Done, 
	Aborted=> , 
	Error=> Service.AutoMode_EmptyBoxMove.HandShake.Error, 
	ErrorID=> , 
	Status=> , 
	UniqueErrorCode=> , 
	INPUT:= INPUT, 
	Cylinder:= Cylinder, 
	Motor:= Motor, 
	Cylinders :=OutRobotCylinders.Cylinders,
	Clips := OutRobotClips.Cylinders,
	AutoMode_OutRobotMoveMove:=Service.AutoMode_EmptyBoxMove ,
	Pause := bStopMem);

fbOutRobot_RareBoxMove(
	Execute:= Service.AutoMode_RareBoxMove.HandShake.Execute ,
	Abort:= THIS^.Abort OR _bAnyServiceError,
	Reset:= Reset,
	ObjectName:= 'fbOutRobot_RareBoxMove', 
	Busy=> Service.AutoMode_RareBoxMove.HandShake.Busy, 
	Done=> Service.AutoMode_RareBoxMove.HandShake.Done, 
	Aborted=> , 
	Error=> Service.AutoMode_RareBoxMove.HandShake.Error, 
	ErrorID=> , 
	Status=> , 
	UniqueErrorCode=> , 
	INPUT:=INPUT , 
	Cylinder:= Cylinder, 
	Motor:= Motor, 
	Cylinders :=OutRobotCylinders.Cylinders,
	Clips := OutRobotClips.Cylinders,
	AutoMode_OutRobotMoveMove:= Service.AutoMode_RareBoxMove,
	Pause := bStopMem);

fbOutRobot_BoxMoveReverse(
	Execute:= Service.AutoMode_BoxMoveReverse.HandShake.Execute,
	Abort:= THIS^.Abort OR _bAnyServiceError,
	Reset:= Reset,
	ObjectName:='fbOutRobot_BoxMoveReverse', 
	Busy=> Service.AutoMode_BoxMoveReverse.HandShake.Busy, 
	Done=> Service.AutoMode_BoxMoveReverse.HandShake.Done, 
	Aborted=> , 
	Error=> Service.AutoMode_BoxMoveReverse.HandShake.Error, 
	ErrorID=> , 
	Status=> , 
	UniqueErrorCode=> , 
	INPUT:= INPUT, 
	Cylinder:= Cylinder, 
	Motor:= Motor, 
	Cylinders :=OutRobotCylinders.Cylinders,
	Clips := OutRobotClips.Cylinders,
	AutoMode_OutRobotMoveMove:= Service.AutoMode_BoxMoveReverse,
	pause := bStopMem);	
	
fbDifferentCVCamera(
	xDone=> Service.AutoMode_DifferentCVCamera.Status.Done,
	xBusy=> Service.AutoMode_DifferentCVCamera.Status.Busy,
	xError=> Service.AutoMode_DifferentCVCamera.Status.Error,
	xExecute:= Service.AutoMode_DifferentCVCamera.Command.Execute,
	xAbort:= Service.AutoMode_DifferentCVCamera.Command.Abort OR THIS^.Abort OR _bAnyServiceError,
	xReset:= Reset,
	Cylinder:= Cylinder, 
	TimeOut:= , 
	Input:= INPUT, 
	OutPut:= OutPut ,
	Motor:= Motor, 
	BoxCameraDone:= Service.AutoMode_DifferentCVCamera.BoxCameraDone, 
	xAborted=> , 
	iErrorID=> , 
	ErrorMsg=> , 
	UseBoxCamera=> Service.AutoMode_DifferentCVCamera.UseBoxCamera);

fbOutRobot_TurnTableToRoundBelt(
	Execute:= fbOutRobot_TurnTableToRoundBel_Ctrl.Execute,
	Abort:= fbOutRobot_TurnTableToRoundBel_Ctrl.Abort OR THIS^.Abort OR _bAnyServiceError,
	Reset:= Reset,
	ObjectName:= 'fbOutRobot_TurnTableToRoundBelt', 
	Busy=> fbOutRobot_TurnTableToRoundBel_Status.Busy, 
	Done=> fbOutRobot_TurnTableToRoundBel_Status.Done, 
	Aborted=> , 
	Error=> fbOutRobot_TurnTableToRoundBel_Status.Error, 
	ErrorID=> , 
	Status=> fbOutRobot_TurnTableToRoundBel_Status.Status, 
	UniqueErrorCode=> , 
	INPUT:= INPUT, 
	Cylinders:= OutRobotCylinders.Cylinders, 
	Clips:=OutRobotClips.Cylinders , 
	AutoMode_TurnTableToRoundBelt:= ); // todo creative var to fill in cmooand info	
	
	fbSameSizeCVCamera(
		xReset := Reset,
		xDone=> Service.AutoMode_SameSizeCVCamera.Status.Done,
		xBusy=> Service.AutoMode_SameSizeCVCamera.Status.Busy,
		xError=> Service.AutoMode_SameSizeCVCamera.Status.Error,
		xExecute:= Service.AutoMode_SameSizeCVCamera.Command.Execute,
		xAbort:= Service.AutoMode_SameSizeCVCamera.Command.Abort OR THIS^.Abort OR _bAnyServiceError,
		Cylinder:= Cylinder, 
		TimeOut:= , 
		Input:= INPUT, 
		OutPut:= OUTPUT, 
		Motor:= Motor, 
		BoxCameraDone:= Service.AutoMode_SameSizeCVCamera.BoxCameraDone, 
		xAborted=> , 
		iErrorID=> , 
		ErrorMsg=> , 
		UseBoxCamera=> Service.AutoMode_SameSizeCVCamera.UseBoxCamera);
		
	fbSameSizeCVCamera_Reverse(
		xReset := Service.AutoMode_SameSizeCVCamera_Reverse.Command.Reset,
		xDone=> Service.AutoMode_SameSizeCVCamera_Reverse.Status.Done,
		xBusy=> Service.AutoMode_SameSizeCVCamera_Reverse.Status.Busy,
		xError=> Service.AutoMode_SameSizeCVCamera_Reverse.Status.Error,
		xExecute:= Service.AutoMode_SameSizeCVCamera_Reverse.Command.Execute,
		xAbort:= Service.AutoMode_SameSizeCVCamera_Reverse.Command.Abort OR THIS^.Abort OR _bAnyServiceError,
		Cylinder:= Cylinder,
		TimeOut:= ,
		Input:= INPUT,
		OutPut:= OUTPUT,
		Motor:= Motor,
		SameSizeCVRequest:= SameSizeCVRequest,
		BoxCameraDone:= Service.AutoMode_SameSizeCVCamera_Reverse.BoxCameraDone,
		xAborted=> ,
		iErrorID=> ,
		ErrorMsg=> ,
		UseBoxCamera=> Service.AutoMode_SameSizeCVCamera_Reverse.UseBoxCamera);
		
	// ================================================================
	// 逆向拍照批次入料 — 逐欄位 link ADS HandShake
	// ================================================================

	// --- fbReverseBoxToWareHouse (子FB: 軌道→大手臂→入倉/NG，輸送帶要先動) ---
	fbReverseBoxToWareHouse(
		// Command (C# → PLC)
		Execute := Service.AutoMode_ReverseBoxToWareHouse.Command.Execute,
		Abort := Service.AutoMode_ReverseBoxToWareHouse.Command.Abort OR THIS^.Abort OR _bAnyServiceError,
		Reset := Service.AutoMode_ReverseBoxToWareHouse.Command.Reset,
		ObjectName := 'Reverse box to warehouse',
		// 盒子資訊 (C# → PLC) — 介面變更:eBoxA/B_Destination enum 三選一 (WareHouse / PullOut / NGConveyor) + 新增 iBoxA/B_PullOutSide
		bBoxA_Enable := Service.AutoMode_ReverseBoxToWareHouse.bBoxA_Enable,
		eBoxA_Destination := Service.AutoMode_ReverseBoxToWareHouse.eBoxA_Destination,
		iBoxA_Warehouse := Service.AutoMode_ReverseBoxToWareHouse.iBoxA_Warehouse,
		iBoxA_Level := Service.AutoMode_ReverseBoxToWareHouse.iBoxA_Level,
		iBoxA_Track := Service.AutoMode_ReverseBoxToWareHouse.iBoxA_Track,
		iBoxA_PullOutSide := Service.AutoMode_ReverseBoxToWareHouse.iBoxA_PullOutSide,
		bBoxB_Enable := Service.AutoMode_ReverseBoxToWareHouse.bBoxB_Enable,
		eBoxB_Destination := Service.AutoMode_ReverseBoxToWareHouse.eBoxB_Destination,
		iBoxB_Warehouse := Service.AutoMode_ReverseBoxToWareHouse.iBoxB_Warehouse,
		iBoxB_Level := Service.AutoMode_ReverseBoxToWareHouse.iBoxB_Level,
		iBoxB_Track := Service.AutoMode_ReverseBoxToWareHouse.iBoxB_Track,
		iBoxB_PullOutSide := Service.AutoMode_ReverseBoxToWareHouse.iBoxB_PullOutSide,
		// 硬體
		Cylinder := Cylinder,
		Motor := Motor,
		SameSizeCVRequest := SameSizeCVRequest,
		Input := INPUT,
		OutPut := OUTPUT,
		StorageRobot := DAS_CoreSys.MachineControl.FanucRobot.List.StorageRobot,
		WareHouse := DAS_CoreSys.MachineControl.fbStorageArea.fbWarehouse,
		PullOutConveyor := fbPulloutCV,
		Stop := bStopMem,
		// Status output (PLC → C#)
		bBoxA_Done => Service.AutoMode_ReverseBoxToWareHouse.bBoxA_Done,
		bBoxB_Done => Service.AutoMode_ReverseBoxToWareHouse.bBoxB_Done);
	// Status (PLC → C#)
	Service.AutoMode_ReverseBoxToWareHouse.Status.Done	:= fbReverseBoxToWareHouse.Done;
	Service.AutoMode_ReverseBoxToWareHouse.Status.Busy	:= fbReverseBoxToWareHouse.Busy;
	Service.AutoMode_ReverseBoxToWareHouse.Status.Error	:= fbReverseBoxToWareHouse.Error;	

	// --- fbReverseBatchPickAndPhoto (主FB: 三軌 Pipeline) ---
	fbReverseBatchPickAndPhoto(
		// Command (C# → PLC)
		Execute := Service.AutoMode_ReverseBatchPick.Command.Execute,
		Abort := Service.AutoMode_ReverseBatchPick.Command.Abort OR THIS^.Abort OR _bAnyServiceError,
		Reset := Service.AutoMode_ReverseBatchPick.Command.Reset,
		ObjectName := 'Reverse batch pick and photo',
		// 鐵盤 Sensor (C# → PLC, 後續改硬體訊號)
		bLeftPlateReady := Service.AutoMode_ReverseBatchPick.bLeftPlateReady,
		bRightPlateReady := Service.AutoMode_ReverseBatchPick.bRightPlateReady,
		// 鐵盤配置 (C# → PLC)
		LeftPlate := Service.AutoMode_ReverseBatchPick.LeftPlate,
		RightPlate := Service.AutoMode_ReverseBatchPick.RightPlate,
		bLeftConfigReady := Service.AutoMode_ReverseBatchPick.bLeftConfigReady,
		bRightConfigReady := Service.AutoMode_ReverseBatchPick.bRightConfigReady,
		// 拍照結果 (C# → PLC)
		BoxCameraDone := Service.AutoMode_ReverseBatchPick.BoxCameraDone,
		CameraIsOK := Service.AutoMode_ReverseBatchPick.CameraIsOK,
		CameraWarehouse := Service.AutoMode_ReverseBatchPick.CameraWarehouse,
		CameraLevel := Service.AutoMode_ReverseBatchPick.CameraLevel,
		CameraTrack := Service.AutoMode_ReverseBatchPick.CameraTrack,
		// 硬體
		Cylinder := Cylinder,
		Motor := Motor,
		SameSizeCVRequest := SameSizeCVRequest,
		Input := INPUT,
		OutPut := OUTPUT,
		StorageRobot := DAS_CoreSys.MachineControl.FanucRobot.List.StorageRobot,
		ShippingRobot := DAS_CoreSys.MachineControl.FanucRobot.List.ShippingRobot,
		WareHouse := DAS_CoreSys.MachineControl.fbStorageArea.fbWarehouse,
		Stop := bStopMem,
		// Status output (PLC → C#)
		bLeftPlateArrived => Service.AutoMode_ReverseBatchPick.bLeftPlateArrived,
		bRightPlateArrived => Service.AutoMode_ReverseBatchPick.bRightPlateArrived,
		bLeftPlateDone => Service.AutoMode_ReverseBatchPick.bLeftPlateDone,
		bRightPlateDone => Service.AutoMode_ReverseBatchPick.bRightPlateDone,
		UseBoxCamera => Service.AutoMode_ReverseBatchPick.UseBoxCamera,
		uiUnphotographedCount => Service.AutoMode_ReverseBatchPick.uiUnphotographedCount,
		uiTotalProcessed => Service.AutoMode_ReverseBatchPick.uiTotalProcessed,
		uiTransportedCount => Service.AutoMode_ReverseBatchPick.uiTransportedCount);
	// Status (PLC → C#)
	Service.AutoMode_ReverseBatchPick.Status.Done	:= fbReverseBatchPickAndPhoto.Done;
	Service.AutoMode_ReverseBatchPick.Status.Busy	:= fbReverseBatchPickAndPhoto.Busy;
	Service.AutoMode_ReverseBatchPick.Status.Error	:= fbReverseBatchPickAndPhoto.Error;

	
fbPulloutCV(
	Execute:= _AutoPullout_Ctrl.Execute,
	Abort:= _AutoPullout_Ctrl.Abort OR THIS^.Abort OR _bAnyServiceError,
	Reset:= Reset,
	ObjectName:= ' Pullout conveyor ', 
	Busy=> _AutoPullout_Status.Busy, 
	Done=> _AutoPullout_Status.Done, 
	Aborted=> , 
	Error=> _AutoPullout_Status.Error, 
	ErrorID=> , 
	Status=> _AutoPullout_Status.Status, 
	UniqueErrorCode=> , 
	FixCylinderA1:= Cylinder.List.fbPullOutCV_AsidePress1, 
	FixCylinderA2:= Cylinder.List.fbPullOutCV_AsidePress2, 
	FixCylinderB1:= Cylinder.List.fbPullOutCV_BsidePress1, 
	FixCylinderB2:= Cylinder.List.fbPullOutCV_BsidePress2, 
	BarrierCylinderA:= Cylinder.List.fbPullOutCV_AsideBlock, 
	BarrierCylinderB:= Cylinder.List.fbPullOutCV_BsideBlock, 
	ConveyorMotorA:= Motor.List.PullOutCV_A, 
	ConveyorMotorB:= Motor.List.PullOutCV_B, 
	INPUT:= INPUT, 
	PullOutInfo:= _AutoPullout_Info);
	
fbPulloutCV_BTNCtrl(
	Input:= INPUT, 
	Output:= OUTPUT, 
	Motor:= Motor, 
	bPullOutConveyorExecute:= _AutoPullout_Ctrl.Execute, 
	bPullOutConveyorDone:= _AutoPullout_Status.Done, 
	bPullOutConveyorBusy:= _AutoPullout_Status.Busy, 
	StroageRegionMode:= eModeCurrent, 
	PullOutConveyorState=> );
	
fbAllocateRobotNeedlingMove(
	xDone=>  Service.AllocateRobotNeedlingMove.Status.Done,
	xBusy=> Service.AllocateRobotNeedlingMove.Status.Busy,
	xError=> Service.AllocateRobotNeedlingMove.Status.Error,
	xExecute:= Service.AllocateRobotNeedlingMove.Command.Execute,
	xAbort:= Service.AllocateRobotNeedlingMove.Command.Abort OR THIS^.Abort OR _bAnyServiceError,
	TimeOut:= , 
	MovingInfo:= Service.AllocateRobotNeedlingMove.MovingInfo, 
	xAborted=> , 
	iErrorID=> , 
	ErrorMsg=> Service.AllocateRobotNeedlingMove.Status.Status);
END_ACTION

ACTION A01_RoundBeltAccessControl:
CASE RoundBeltControlAccess OF 
	E_RoundBeltControlAccess.Host :
	 IF eModeCurrent = E_UnitMode.Manual THEN
		_RoundBeltMoveJob.Position :=Service.AllocateCircleMove.Position;
		_RoundBeltMoveJob.Latch :=Service.AllocateCircleMove.Latch;
		_RoundBeltMoveJob.HandShake.Execute :=Service.AllocateCircleMove.HandShake.Execute;
		_RoundBeltMoveJob.HandShake.Reset :=Service.AllocateCircleMove.HandShake.Reset;
		_RoundBeltMoveJob.HandShake.Occupied  :=Service.AllocateCircleMove.HandShake.Occupied;
		Service.AllocateCircleMove.HandShake.Busy := _RoundBeltMoveJob.HandShake.Busy;
		Service.AllocateCircleMove.HandShake.Done := _RoundBeltMoveJob.HandShake.Done;
		Service.AllocateCircleMove.HandShake.Error := _RoundBeltMoveJob.HandShake.Error;
	ELSIF  eModeCurrent = E_UnitMode.Auto THEN
		_RoundBeltMoveJob.Position :=Service.AutoMode_AllocateCircleMove.Position;
		_RoundBeltMoveJob.Latch :=Service.AutoMode_AllocateCircleMove.Latch;
		_RoundBeltMoveJob.HandShake.Execute :=Service.AutoMode_AllocateCircleMove.HandShake.Execute;
		_RoundBeltMoveJob.HandShake.Reset :=Service.AutoMode_AllocateCircleMove.HandShake.Reset;
		_RoundBeltMoveJob.HandShake.Occupied  :=Service.AutoMode_AllocateCircleMove.HandShake.Occupied;
		Service.AutoMode_AllocateCircleMove.HandShake.Busy := _RoundBeltMoveJob.HandShake.Busy;
		Service.AutoMode_AllocateCircleMove.HandShake.Done := _RoundBeltMoveJob.HandShake.Done;
		Service.AutoMode_AllocateCircleMove.HandShake.Error := _RoundBeltMoveJob.HandShake.Error;
	END_IF
		
	E_RoundBeltControlAccess.Allocating  :
	
		_RoundBeltMoveJob.Position :=RoundBeltMoveJob_Position;
		//_RoundBeltMoveJob.Latch :=;
		_RoundBeltMoveJob.HandShake.Execute :=RoundBeltMoveJob_Ctrl_Batch.Execute;
		_RoundBeltMoveJob.HandShake.Reset :=RoundBeltMoveJob_Ctrl_Batch.Reset;
		RoundBeltMoveJob_Status.Busy := _RoundBeltMoveJob.HandShake.Busy;
		RoundBeltMoveJob_Status.Done := _RoundBeltMoveJob.HandShake.Done;
		RoundBeltMoveJob_Status.Error := _RoundBeltMoveJob.HandShake.Error;

	E_RoundBeltControlAccess.FanucRobot:
		_RoundBeltMoveJob.Position :=RoundBeltMoveJob_Position_FanucRobot;
		//_RoundBeltMoveJob.Latch :=;
		_RoundBeltMoveJob.HandShake.Execute :=RoundBeltMoveJob_Ctrl.Execute;
		_RoundBeltMoveJob.HandShake.Reset :=RoundBeltMoveJob_Ctrl.Reset;
		RoundBeltMoveJob_Status.Busy := _RoundBeltMoveJob.HandShake.Busy;
		RoundBeltMoveJob_Status.Done := _RoundBeltMoveJob.HandShake.Done;
		RoundBeltMoveJob_Status.Error := _RoundBeltMoveJob.HandShake.Error;	
END_CASE
END_ACTION

ACTION A02_PulloutAccessControl:
CASE PulloutControlAccess OF
    E_RoundBeltControlAccess.Host:
        _AutoPullout_Ctrl.Execute := Service.AutoMode_PullOutConveyor.Command.Execute;
        _AutoPullout_Ctrl.Abort := Service.AutoMode_PullOutConveyor.Command.Abort;
        _AutoPullout_Ctrl.Reset := Service.AutoMode_PullOutConveyor.Command.Reset;
        Service.AutoMode_PullOutConveyor.Status.Busy := _AutoPullout_Status.Busy;
        Service.AutoMode_PullOutConveyor.Status.Done := _AutoPullout_Status.Done;
        Service.AutoMode_PullOutConveyor.Status.Error := _AutoPullout_Status.Error;
        Service.AutoMode_PullOutConveyor.Status.Status := _AutoPullout_Status.Status;
        _AutoPullout_Info := Service.AutoMode_PullOutConveyor.PullOutConveyorInfo;
    E_RoundBeltControlAccess.Allocating:
        _AutoPullout_Ctrl.Execute := AutoPullout_Internal_Ctrl.Execute;
        _AutoPullout_Ctrl.Abort := AutoPullout_Internal_Ctrl.Abort;
        _AutoPullout_Ctrl.Reset := AutoPullout_Internal_Ctrl.Reset;
        AutoPullout_Internal_Status.Busy := _AutoPullout_Status.Busy;
        AutoPullout_Internal_Status.Done := _AutoPullout_Status.Done;
        AutoPullout_Internal_Status.Error := _AutoPullout_Status.Error;
        AutoPullout_Internal_Status.Status := _AutoPullout_Status.Status;
        _AutoPullout_Info := AutoPullout_Internal_Info;
    E_RoundBeltControlAccess.FanucRobot:
        _AutoPullout_Ctrl.Execute := RobotPullout_Internal_Ctrl.Execute;
        _AutoPullout_Ctrl.Abort := RobotPullout_Internal_Ctrl.Abort;
        _AutoPullout_Ctrl.Reset := RobotPullout_Internal_Ctrl.Reset;
        RobotPullout_Internal_Status.Busy := _AutoPullout_Status.Busy;
        RobotPullout_Internal_Status.Done := _AutoPullout_Status.Done;
        RobotPullout_Internal_Status.Error := _AutoPullout_Status.Error;
        RobotPullout_Internal_Status.Status := _AutoPullout_Status.Status;
        _AutoPullout_Info := RobotPullout_Internal_Info;
END_CASE
END_ACTION

ACTION A99_ErrorHandler:

END_ACTION

METHOD M_Aborted
Abort := FALSE;
M_StateComplete();
END_METHOD

METHOD M_Aborting
Abort := TRUE;
M_StateComplete();
END_METHOD

METHOD M_ActiveRoundBeltInternalCtrl : BOOL
VAR_INPUT
END_VAR
bReloadRotateBeltRequest := TRUE;
M_ActiveRoundBeltInternalCtrl := true; // Method end
END_METHOD

METHOD PRIVATE M_AutoAllocatingBatch : BOOL
VAR_INPUT
END_VAR
IF NOT Service.AutoMode_SimpleAllocation_Batch.HandShake.Execute 
   AND NOT Service.AutoMode_SimpleAllocation_Batch.HandShake.Busy
   AND NOT Service.AutoMode_AllocateBatchMode_Reverse.HandShake.Execute
   AND NOT Service.AutoMode_AllocateBatchMode_Reverse.HandShake.Busy THEN
	
	AutoAllocateJobBatch_Ctrl.bSimpleAllocation:=FALSE;
	AutoAllocateJobBatch_Ctrl.bExecute:=Service.AutoMode_AllocateBatchMode.HandShake.Execute;
	AutoAllocateJobBatch_Ctrl.bReset :=Service.AutoMode_AllocateBatchMode.HandShake.Reset;
	AutoAllocateJobBatch_Ctrl.bOccupied:=Service.AutoMode_AllocateBatchMode.HandShake.Occupied;
	AutoAllocateJobBatch_Ctrl.bPause :=Service.AutoMode_AllocateBatchMode.Pause;

	AutoAllocateJobBatch_Ctrl.AutoMode_AllocateMoveBatch.AllocationInfo:=Service.AutoMode_AllocateBatchMode.AllocationInfo;
	AutoAllocateJobBatch_Ctrl.AutoMode_AllocateMoveBatch.NrOfAllocationJob:=Service.AutoMode_AllocateBatchMode.NrOfAllocationJob;

	Service.AutoMode_AllocateBatchMode.WorkedID:=AutoAllocateJobBatch_Ctrl.AutoMode_AllocateMoveBatch.WorkedID;
	Service.AutoMode_AllocateBatchMode.HandShake.Busy:= AutoAllocateJobBatch_Status.bBusy;
	Service.AutoMode_AllocateBatchMode.HandShake.Error:= AutoAllocateJobBatch_Status.bError;
	Service.AutoMode_AllocateBatchMode.HandShake.Done:= AutoAllocateJobBatch_Status.bDone;
	
	RoundBeltMoveJob_Ctrl_Batch :=fb_AllocateBatchMode.RoundBeltMoveJob_Ctrl; 
	RoundBeltMoveJob_Position :=fb_AllocateBatchMode.RoundBeltMoveJob_Position;	
	bAutoAllocateJobDryRun := FALSE;
END_IF
END_METHOD

METHOD PRIVATE M_AutoAllocatingBatch_Reverse : BOOL
VAR_INPUT
END_VAR
IF NOT Service.AutoMode_AllocateBatchMode.HandShake.Execute 
   AND NOT Service.AutoMode_AllocateBatchMode.HandShake.Busy
   AND NOT Service.AutoMode_SimpleAllocation_Batch.HandShake.Execute
   AND NOT Service.AutoMode_SimpleAllocation_Batch.HandShake.Busy THEN
	AutoAllocateJobBatch_Reverse_Ctrl.bExecute:=Service.AutoMode_AllocateBatchMode_Reverse.HandShake.Execute;
	AutoAllocateJobBatch_Reverse_Ctrl.bReset :=Service.AutoMode_AllocateBatchMode_Reverse.HandShake.Reset;
	AutoAllocateJobBatch_Reverse_Ctrl.bOccupied:=Service.AutoMode_AllocateBatchMode_Reverse.HandShake.Occupied;
	AutoAllocateJobBatch_Reverse_Ctrl.bPause :=Service.AutoMode_AllocateBatchMode_Reverse.Pause;

	AutoAllocateJobBatch_Reverse_Ctrl.AutoMode_AllocateMoveBatch.AllocationInfo:=Service.AutoMode_AllocateBatchMode_Reverse.AllocationInfo;
	AutoAllocateJobBatch_Reverse_Ctrl.AutoMode_AllocateMoveBatch.NrOfAllocationJob:=Service.AutoMode_AllocateBatchMode_Reverse.NrOfAllocationJob;

	Service.AutoMode_AllocateBatchMode_Reverse.WorkedID:=AutoAllocateJobBatch_Reverse_Ctrl.AutoMode_AllocateMoveBatch.WorkedID;
	Service.AutoMode_AllocateBatchMode_Reverse.HandShake.Busy:= AutoAllocateJobBatch_Reverse_Status.bBusy;
	Service.AutoMode_AllocateBatchMode_Reverse.HandShake.Error:= AutoAllocateJobBatch_Reverse_Status.bError;
	Service.AutoMode_AllocateBatchMode_Reverse.HandShake.Done:= AutoAllocateJobBatch_Reverse_Status.bDone;
	RoundBeltMoveJob_Ctrl_Batch :=fb_AllocateBatchMode_Reverse.RoundBeltMoveJob_Ctrl; 
	RoundBeltMoveJob_Position :=fb_AllocateBatchMode_Reverse.RoundBeltMoveJob_Position;	

	bAutoAllocateJobDryRun := FALSE;
	
	END_IF
END_METHOD

METHOD PRIVATE M_AutoAllocatingBatch_Simple : BOOL
VAR_INPUT
END_VAR
IF NOT Service.AutoMode_AllocateBatchMode.HandShake.Execute 
   AND NOT Service.AutoMode_AllocateBatchMode.HandShake.Busy
   AND NOT Service.AutoMode_AllocateBatchMode_Reverse.HandShake.Execute
   AND NOT Service.AutoMode_AllocateBatchMode_Reverse.HandShake.Busy THEN
	
	AutoAllocateJobBatch_Ctrl.bSimpleAllocation:=TRUE;
	AutoAllocateJobBatch_Ctrl.bExecute:=Service.AutoMode_SimpleAllocation_Batch.HandShake.Execute;
	AutoAllocateJobBatch_Ctrl.bReset :=Service.AutoMode_SimpleAllocation_Batch.HandShake.Reset;
	AutoAllocateJobBatch_Ctrl.bOccupied:=Service.AutoMode_SimpleAllocation_Batch.HandShake.Occupied;
	AutoAllocateJobBatch_Ctrl.bPause :=Service.AutoMode_SimpleAllocation_Batch.Pause;

	AutoAllocateJobBatch_Ctrl.AutoMode_AllocateMoveBatch.AllocationInfo:=Service.AutoMode_SimpleAllocation_Batch.AllocationInfo;
	AutoAllocateJobBatch_Ctrl.AutoMode_AllocateMoveBatch.NrOfAllocationJob:=Service.AutoMode_SimpleAllocation_Batch.NrOfAllocationJob;

	Service.AutoMode_SimpleAllocation_Batch.WorkedID:=AutoAllocateJobBatch_Ctrl.AutoMode_AllocateMoveBatch.WorkedID;
	Service.AutoMode_SimpleAllocation_Batch.HandShake.Busy:= AutoAllocateJobBatch_Status.bBusy;
	Service.AutoMode_SimpleAllocation_Batch.HandShake.Error:= AutoAllocateJobBatch_Status.bError;
	Service.AutoMode_SimpleAllocation_Batch.HandShake.Done:= AutoAllocateJobBatch_Status.bDone;
	
	RoundBeltMoveJob_Ctrl_Batch :=fb_AllocateBatchMode.RoundBeltMoveJob_Ctrl; 
	RoundBeltMoveJob_Position :=fb_AllocateBatchMode.RoundBeltMoveJob_Position;		

	bAutoAllocateJobDryRun := FALSE;
END_IF
END_METHOD

METHOD PRIVATE M_AutoTurnTable : BOOL
VAR_INPUT
END_VAR
_TurnTableMove.HandShake.Execute:=Service.AutoMode_TurnTableMove.HandShake.Execute;
_TurnTableMove.Position:=Service.AutoMode_TurnTableMove.Position;

Service.AutoMode_TurnTableMove.HandShake.Busy := _TurnTableMove.HandShake.Busy;
Service.AutoMode_TurnTableMove.HandShake.Done := _TurnTableMove.HandShake.Done;
Service.AutoMode_TurnTableMove.HandShake.Error := _TurnTableMove.HandShake.Error;
END_METHOD

METHOD PRIVATE M_CheckAxesHomed : BOOL
VAR_INPUT
END_VAR

VAR 
	AxisIndex : INT;//1-6
	bCheckHome : BOOL:=TRUE;
END_VAR
bCheckHome:=TRUE;

FOR AxisIndex :=1 TO 6 DO
	bCheckHome:=bCheckHome AND	arAxisCtrl_gb[AxisIndex].Admin.Axis.Status.Homed;
END_FOR

M_CheckAxesHomed:=	bCheckHome;
END_METHOD

METHOD M_Clearing
M_StateComplete();
END_METHOD

METHOD M_Complete
M_StateComplete();
END_METHOD

METHOD M_Completing
M_StateComplete();
END_METHOD

METHOD M_Execute
CASE eModeCurrent OF
	E_UnitMode.Manual:
		M_ManualAllocating();
		M_AutoAllocatingBatch_Simple();
		M_AutoAllocatingBatch();
		M_AutoAllocatingBatch_Reverse();
		M_ManualTurnTable();
		M_AutoAllocatingBatch_Reverse();
		//M_TransCVCameraPress_ManualMode();
		//TransCV_Press :=FALSE;

	E_UnitMode.Auto:
	
		M_AutoAllocatingBatch_Simple();
		M_AutoAllocatingBatch();
		M_AutoAllocatingBatch_Reverse();
		M_AutoTurnTable();
		M_TransCVCameraPress();
END_CASE
//M_StateComplete();
A00_Service();
A01_RoundBeltAccessControl();
A02_PulloutAccessControl();
//bHomed :=M_CheckAxesHomed();
END_METHOD

METHOD PUBLIC M_GetPulloutAccess : BOOL
VAR_INPUT
	 ControlAccess:	 E_RoundBeltControlAccess;
END_VAR
IF THIS^.PulloutControlAccess = E_RoundBeltControlAccess.Host AND 
	NOT (fbPulloutCV.Execute OR fbPulloutCV.Busy OR fbPulloutCV.Done) THEN
	THIS^.PulloutControlAccess := ControlAccess;
	M_GetPulloutAccess := TRUE;
 ELSE
	M_GetPulloutAccess := FALSE;	
 END_IF
END_METHOD

METHOD PUBLIC M_GetRoundBeltAccess : BOOL
VAR_INPUT
	 ControlAccess:	 E_RoundBeltControlAccess;
END_VAR
IF THIS^.RoundBeltControlAccess = E_RoundBeltControlAccess.Host AND 
	NOT (RoundBeltControl.xExecute OR RoundBeltControl.xBusy OR RoundBeltControl.xDone) THEN
	THIS^.RoundBeltControlAccess := ControlAccess;
	M_GetRoundBeltAccess := TRUE;
 ELSE
	M_GetRoundBeltAccess := FALSE;	
 END_IF
END_METHOD

METHOD M_Held
M_StateComplete();
END_METHOD

METHOD M_Holding
M_StateComplete();
END_METHOD

METHOD M_Idle
M_StateComplete();
END_METHOD

METHOD M_InactiveRoundBeltInternalCtrl : BOOL
VAR_INPUT
END_VAR
bReloadRotateBeltRequest := FALSE;

M_InactiveRoundBeltInternalCtrl := true; // Method end
END_METHOD

METHOD PRIVATE M_ManualAllocating : BOOL
VAR_INPUT
END_VAR

VAR_INST 
	
END_VAR

	AutoAllocateJobBatch_Ctrl.bSimpleAllocation:=FALSE;
	AutoAllocateJobBatch_Ctrl.bReset:=Service.AllocateMoveStructure.HandShake.Reset;
	AutoAllocateJobBatch_Ctrl.bPause:=FALSE;
	AutoAllocateJobBatch_Ctrl.bOccupied :=Service.AllocateMoveStructure.HandShake.Occupied;
	AutoAllocateJobBatch_Ctrl.bExecute:=Service.AllocateMoveStructure.HandShake.Execute;
	AutoAllocateJobBatch_Ctrl.AutoMode_AllocateMoveBatch.NrOfAllocationJob:=1;
	AutoAllocateJobBatch_Ctrl.AutoMode_AllocateMoveBatch.AllocationInfo[0].FastMode:=FALSE;
	AutoAllocateJobBatch_Ctrl.AutoMode_AllocateMoveBatch.AllocationInfo[0].SyncMode:=FALSE	;
	
	AutoAllocateJobBatch_Ctrl.AutoMode_AllocateMoveBatch.AllocationInfo[0].PickingNeedleInfo[0].CycleStart:=TRUE;
	AutoAllocateJobBatch_Ctrl.AutoMode_AllocateMoveBatch.AllocationInfo[0].PickingNeedleInfo[0].Box:=LREAL_TO_UINT( Service.AllocateMoveStructure.Frombox);
	AutoAllocateJobBatch_Ctrl.AutoMode_AllocateMoveBatch.AllocationInfo[0].PickingNeedleInfo[0].Clip:=LREAL_TO_INT(Service.AllocateMoveStructure.Clip);
	AutoAllocateJobBatch_Ctrl.AutoMode_AllocateMoveBatch.AllocationInfo[0].PickingNeedleInfo[0].NeedleLocation:=LREAL_TO_INT(Service.AllocateMoveStructure.FromPosition);
	AutoAllocateJobBatch_Ctrl.AutoMode_AllocateMoveBatch.AllocationInfo[0].PlacingNeedleInfo[0].CycleStart:=TRUE;
	
	AutoAllocateJobBatch_Ctrl.AutoMode_AllocateMoveBatch.AllocationInfo[0].PlacingNeedleInfo[0].Box :=LREAL_TO_UINT(Service.AllocateMoveStructure.Tobox);
	AutoAllocateJobBatch_Ctrl.AutoMode_AllocateMoveBatch.AllocationInfo[0].PlacingNeedleInfo[0].Clip:=LREAL_TO_INT(Service.AllocateMoveStructure.Clip);
	AutoAllocateJobBatch_Ctrl.AutoMode_AllocateMoveBatch.AllocationInfo[0].PlacingNeedleInfo[0].NeedleLocation :=LREAL_TO_INT(Service.AllocateMoveStructure.ToPosition);

	Service.AllocateMoveStructure.HandShake.Busy :=AutoAllocateJobBatch_Status.bBusy;
	Service.AllocateMoveStructure.HandShake.Done :=AutoAllocateJobBatch_Status.bDone;
	Service.AllocateMoveStructure.HandShake.Error :=AutoAllocateJobBatch_Status.bError;
	bAutoAllocateJobDryRun := TRUE;
END_METHOD

METHOD PRIVATE M_ManualTurnTable : BOOL
VAR_INPUT
END_VAR
_TurnTableMove.HandShake.Execute:=Service.TurnTableMove.HandShake.Execute;
_TurnTableMove.Position:=Service.TurnTableMove.Position;

Service.TurnTableMove.HandShake.Busy := _TurnTableMove.HandShake.Busy;
Service.TurnTableMove.HandShake.Done := _TurnTableMove.HandShake.Done;
Service.TurnTableMove.HandShake.Error := _TurnTableMove.HandShake.Error;
END_METHOD

METHOD PUBLIC M_ReleasePulloutAccess : BOOL
VAR_INPUT
 ControlAccess:	 E_RoundBeltControlAccess;
END_VAR
IF ControlAccess = THIS^.PulloutControlAccess THEN
		THIS^.PulloutControlAccess := E_RoundBeltControlAccess.Host;
		M_ReleasePulloutAccess := TRUE;
	ELSE
		M_ReleasePulloutAccess := FALSE;
	
END_IF
END_METHOD

METHOD PUBLIC M_ReleaseRoundBeltAccess : BOOL
VAR_INPUT
 ControlAccess:	 E_RoundBeltControlAccess;
END_VAR
IF ControlAccess = THIS^.RoundBeltControlAccess THEN
		THIS^.RoundBeltControlAccess := E_RoundBeltControlAccess.Host;
		M_ReleaseRoundBeltAccess := TRUE;
	ELSE
		M_ReleaseRoundBeltAccess := FALSE;
	
END_IF
END_METHOD

METHOD M_ResetReloadRoundBeltAction : BOOL
VAR_INPUT
END_VAR
RoundBeltMoveJob_Ctrl.Execute := FALSE;

M_ResetReloadRoundBeltAction := true; // Method end
END_METHOD

METHOD M_Resetting
IF __ISVALIDREF(Cylinder) THEN
	Clip.stCylinders.Cylinder0 REF= Cylinder.List.fbAllocateRobot_LeftClamp1;
	Clip.stCylinders.Cylinder1 REF= Cylinder.List.fbAllocateRobot_LeftClamp2;
	Clip.stCylinders.Cylinder2 REF= Cylinder.List.fbAllocateRobot_RightClamp1;
	Clip.stCylinders.Cylinder3 REF= Cylinder.List.fbAllocateRobot_RightClamp2;
	Cylinders.stCylinders.Cylinder0 REF= Cylinder.List.fbAllocateRobot_LeftVert1;
	Cylinders.stCylinders.Cylinder1 REF= Cylinder.List.fbAllocateRobot_LeftVert2;
	Cylinders.stCylinders.Cylinder2 REF= Cylinder.List.fbAllocateRobot_RightVert1;
	Cylinders.stCylinders.Cylinder3 REF= Cylinder.List.fbAllocateRobot_RightVert2;	
END_IF

M_StateComplete();
END_METHOD

METHOD PUBLIC M_StartAllocatePulloutAction : BOOL
VAR_INPUT
	CV_ForwardTime :TIME;
	CV_BackwardTIme : TIME;
	CommandType : E_PullOutConveyorCommandType; // Select PullOut conveyor command.
END_VAR
AutoPullout_Internal_Ctrl.Execute := TRUE;
AutoPullout_Internal_Info.ConveyorReverseTime := CV_BackwardTIme;
AutoPullout_Internal_Info.ConveyorRunningTime := CV_ForwardTime;
AutoPullout_Internal_Info.CommandType := CommandType;
M_StartAllocatePulloutAction := TRUE; // Method end
END_METHOD

METHOD M_StartHoming
VAR_INPUT
END_VAR
fbAllocateHome.xExecute := true;
END_METHOD

METHOD M_Starting
M_StateComplete();
END_METHOD

(* This Method is used to start round belt action : unlock pin and move to target position
	also injection the action parameter.
*)
METHOD M_StartReloadRoundBeltAtion : BOOL
VAR_INPUT
	ReloadStation : E_RoundBeltStation;
END_VAR
VAR_INST
	_ReloadStation : E_RoundBeltStation;
END_VAR
IF (ReloadStation > 12) THEN
	_ReloadStation := (ReloadStation -12 );
//	_ReloadStation := (ReloadStation -6 );
ELSE
	_ReloadStation := ReloadStation + 28;
END_IF
IF F_Even(_ReloadStation) THEN
	_ReloadStation := _ReloadStation-1;
END_IF

//IF ReloadStation > 6 THEN
//	_ReloadStation := ReloadStation -6;
//ELSE
//	_ReloadStation := ReloadStation +14;
//END_IF
//AutoRotatebelt_Internal_Ctrl.uiLatch := E_Pistons.LoadingBoxRegion;
//AutoRotatebelt_Internal_Ctrl.uiStation :=  _ReloadStation;
//AutoRotatebelt_Internal_Ctrl.Timeout := T#15S;
//AutoRotatebelt_Internal_Ctrl.bSendPressBox := FALSE; // Release allocate zone, press box cylinder in backward position
RoundBeltMoveJob_Position_FanucRobot := _ReloadStation;
RoundBeltMoveJob_Ctrl.Execute := TRUE;

M_StartReloadRoundBeltAtion := TRUE; // Method end
END_METHOD

METHOD M_StartStoragePulloutAction : BOOL
VAR_INPUT
	CV_ForwardTime :TIME;
	CV_BackwardTIme : TIME;
	CommandType : E_PullOutConveyorCommandType; // Select PullOut conveyor command.
END_VAR
RobotPullout_Internal_Ctrl.Execute := TRUE;
RobotPullout_Internal_Info.CommandType := CommandType;
RobotPullout_Internal_Info.ConveyorReverseTime := CV_BackwardTIme;
RobotPullout_Internal_Info.ConveyorRunningTime := CV_ForwardTime;
M_StartStoragePulloutAction := TRUE; // Method end
END_METHOD

METHOD M_StopAllocatePulloutAction : BOOL
VAR_INPUT
END_VAR
AutoPullout_Internal_Ctrl.Execute := FALSE;
M_StopAllocatePulloutAction := TRUE; // Methode end
END_METHOD

METHOD M_StopHoming
VAR_INPUT
END_VAR
fbAllocateHome.xExecute := False;
END_METHOD

METHOD M_Stopped
M_StateComplete();
END_METHOD

METHOD M_Stopping
M_StateComplete();
END_METHOD

METHOD M_StopStoragePulloutAction : BOOL
VAR_INPUT
END_VAR
RobotPullout_Internal_Ctrl.Execute := FALSE;
M_StopStoragePulloutAction := TRUE; //Method End
END_METHOD

METHOD M_Suspended
M_StateComplete();
END_METHOD

METHOD M_Suspending
M_StateComplete();
END_METHOD

METHOD PUBLIC M_TransCVCameraPress : BOOL
VAR_INPUT
END_VAR
VAR_INST
	
END_VAR
IF NOT TransCV_Press THEN
	//Cylinder.List.fbSameSizeCV_Press2.M_Extend();
	//Cylinder.List.fbDifferentSizeCV_Press1.M_Extend();
	TransCV_Press:=true;
END_IF
END_METHOD

METHOD PUBLIC M_TransCVCameraPress_ManualMode : BOOL
VAR_INPUT
END_VAR
IF TransCV_Press THEN
TransCV_Press := FALSE;
Cylinder.List.fbSameSizeCV_Press2.M_Retract();
Cylinder.List.fbDifferentSizeCV_Press1.M_Retract();
Cylinder.List.fbUpCV_Block1.M_Retract();
END_IF
END_METHOD

METHOD M_Undefined
M_StateComplete();
END_METHOD

METHOD M_Unholding
M_StateComplete();
END_METHOD

METHOD M_Unsuspending
M_StateComplete();
END_METHOD

END_FUNCTION_BLOCK

// ---- Library/20_MachineUnits/22_AllocateArea/Service/FB_AllocateAreaHome.TcPOU
FUNCTION_BLOCK FB_AllocateAreaHome EXTENDS FB_ActionBasic
VAR_INPUT
    xExecute      : BOOL;
    xAbort        : BOOL;

    Cylinder : REFERENCE TO UNI_CylinderList;
	Motor    : REFERENCE TO UNI_MotorList;
	CurrentData      : ST_SetupPara;
    TimeOut  : LREAL := 90; // Unit : s
	Homed : REFERENCE TO BOOL;
END_VAR
VAR_OUTPUT
    xAborted : BOOL;
    iErrorID : INT;
    ErrorMsg : STRING;
	AxisHomingRequest : BOOL;
END_VAR
VAR
    StateBehavior   : CBML.ETrigATo;
    CurrentPosition : ST_PositionTable;
    uiCyclicStep    : UINT := 0;
    uiIndexLoop     : UINT;
	fbExecuteEdgeDetect :FB_EdgeDetect;
END_VAR

THIS^.IBehaviourModel := StateBehavior;
StateBehavior(xExecute := xExecute,
              xAbort := xAbort OR fbExecuteEdgeDetect.xFallingEdge,
              udiTimeOut := LREAL_TO_UDINT( TimeOut*1000000),
              xDone => xDone,
              xBusy => xBusy,
              xError => xError,
              xAborted => xAborted);	

//Make sure that C# turns off execute to shut down the service
fbExecuteEdgeDetect(xInput :=xExecute);

//Error Msg
iErrorID := StateBehavior._model.iErrorID;
ErrorMsg := M_GetErrorMsg(xErrorID := iErrorID);

METHOD CleanupAction
VAR_INPUT
    xAbortProposed : BOOL;
    iErrorIDProposed: INT;
END_VAR
VAR_OUTPUT
    xComplete : BOOL := TRUE;
    xAbort: BOOL := xAbortProposed;
 	iErrorID : INT := iErrorIDProposed;
END_VAR
uiCyclicStep := 0;
END_METHOD

METHOD CyclicAction
VAR_INPUT
    itfTimingController : CBML.ITimingController;
END_VAR
VAR_OUTPUT
    xComplete : BOOL := TRUE;
    iErrorID : INT := 0;
END_VAR
VAR_INST
	
END_VAR

VAR
	AxisIndex 		: INT ; //1-6
	CylinderIndex 	: INT ;
	MotorIndex		: INT ;// 23-26
	bAxesCheck 		: BOOL;
	bCylinderCheck  : BOOL;
	bHomeCheck 		: BOOL;
	bMotorCheck		: BOOL;
END_VAR
xComplete := FALSE;
CASE uiCyclicStep OF
    0: //Check Motor
		bMotorCheck:= TRUE;
		FOR MotorIndex :=23 TO 26 DO
			bMotorCheck := bMotorCheck AND Motor.arMotor[MotorIndex].InStopped;
			IF Motor.arMotor[MotorIndex].xError THEN
				Motor.arMotor[MotorIndex].M_Reset();
			ELSE
				Motor.arMotor[MotorIndex].M_MotorStop();
			END_IF
		END_FOR
		IF bMotorCheck THEN
			uiCyclicStep:=100;
		END_IF
		
	100: // Check Axes error
		bAxesCheck:=TRUE;
		FOR AxisIndex :=1 TO 6 DO
			bAxesCheck := bAxesCheck AND NOT arAxisCtrl_gb[AxisIndex].Admin.Axis.Status.Error;
			IF arAxisCtrl_gb[AxisIndex].Admin.Axis.Status.Error THEN
				arAxisCtrl_gb[AxisIndex].Admin.ClearError:=TRUE;
			END_IF
		END_FOR
		
		IF bAxesCheck THEN
			uiCyclicStep:=200;
		END_IF
			
	200: // Reset All cylinder
		FOR AxisIndex :=1 TO 6 DO 	arAxisCtrl_gb[AxisIndex].Admin.ClearError:=FALSE;	END_FOR
		bCylinderCheck:=TRUE;
		FOR CylinderIndex:=15 TO 20 DO
			bCylinderCheck:=bCylinderCheck AND NOT Cylinder.arCylinder[CylinderIndex].xError;
			IF Cylinder.arCylinder[CylinderIndex].xError THEN
				Cylinder.arCylinder[CylinderIndex].M_Reset();
			END_IF
		END_FOR
		FOR CylinderIndex:=27 TO 53 DO
			bCylinderCheck:=bCylinderCheck AND NOT Cylinder.arCylinder[CylinderIndex].xError;
			IF Cylinder.arCylinder[CylinderIndex].xError THEN
				Cylinder.arCylinder[CylinderIndex].M_Reset();
			END_IF
		END_FOR
		IF bCylinderCheck THEN
			uiCyclicStep:=300;
		END_IF

	300:
		bCylinderCheck:=TRUE;
		FOR CylinderIndex:=15 TO 20 DO
			bCylinderCheck:=bCylinderCheck AND Cylinder.arCylinder[CylinderIndex].InRearPosition;
			Cylinder.arCylinder[CylinderIndex].M_Retract();
		END_FOR
		FOR CylinderIndex:=27 TO 53 DO
			bCylinderCheck:=bCylinderCheck AND Cylinder.arCylinder[CylinderIndex].InRearPosition;
			Cylinder.arCylinder[CylinderIndex].M_Retract();
		END_FOR
		IF bCylinderCheck THEN
			uiCyclicStep:=400;
		END_IF

	400:
		//bHomeCheck := TRUE;
		//IF DAS_CoreSys.MachineControl.fanucrobot.List.StorageRobot._uo1.UO07_AtPerch THEN
			AxisHomingRequest := TRUE;
			IF NOT arAxisCtrl_gb[AxisNo.TurnTable].Admin.Axis.Status.Homed  THEN
			uiCyclicStep:=500;
		//END_IF
		END_IF
		
		

500:	
		bHomeCheck:=TRUE;
		FOR AxisIndex :=1 TO 6 DO
			bHomeCheck := bHomeCheck AND arAxisStatus_gb[AxisIndex].Admin.CmdDone ;//AND arAxisCtrl_gb[AxisIndex].Admin.Axis.Status.Homed;
		END_FOR
		bHomeCheck := arAxisCtrl_gb[AxisNo.Allocate_X].Admin.Axis.Status.Homed AND
			 arAxisCtrl_gb[AxisNo.OutRobot_X].Admin.Axis.Status.Homed AND 
			 arAxisCtrl_gb[AxisNo.OutRobot_Y].Admin.Axis.Status.Homed AND 
			 arAxisCtrl_gb[AxisNo.RoundBelt].Admin.Axis.Status.Homed AND 
			 arAxisCtrl_gb[AxisNo.TurnTable].Admin.Axis.Status.Homed AND 
			 GVL_Machine.AllocatYAxisHome;

		
		IF bHomeCheck THEN
			uiCyclicStep:=600;
		END_IF
	
	600:
		Homed := TRUE;
		xComplete := TRUE;
END_CASE
END_METHOD

METHOD ExitAction
VAR_INPUT
    xAfterCleanup : BOOL;
    xInCopyCode : BOOL;
END_VAR
END_METHOD

METHOD M_GetErrorMsg : T_MaxString
VAR_INPUT
	xErrorID: INT;
END_VAR

VAR
	
END_VAR
CASE xErrorID OF
	0:
		M_GetErrorMsg := 'No Error';
	1:
		M_GetErrorMsg := 'FB_AllocateAreaHome ErrorID 1: Action time out';
//	2:
//		M_GetErrorMsg := 'Position Data invalid';
//	3:
//		M_GetErrorMsg := 'Index invalid';
//	4:
//		M_GetErrorMsg := 'Axis roundbelt not ready has Error';
//	5:
//		M_GetErrorMsg := 'Cylinder not ready has Error';
//	6:
//		M_GetErrorMsg := 'Axis RoundBelt has Error';
//	7:
//		M_GetErrorMsg := 'ChargeZone_Plug has Error';
//	8:
//		M_GetErrorMsg := 'TransmitCVZone_Plug has Error';
//	9:
//		M_GetErrorMsg := 'WorkZone_Plug has Error';
//	10:
//		M_GetErrorMsg := 'WorkZone_Press has Error';
END_CASE
END_METHOD

METHOD PRIVATE M_SetAllHomePars : BOOL
VAR_INPUT
END_VAR
//Allocate X

arAxisCtrl_gb[AxisNo.Allocate_X].Admin._OpMode.en := ModeHoming;

//Allocate Y
arAxisCtrl_gb[AxisNo.Allocate_Y].Admin._OpMode.en := ModePosAbs;

//OutRobot X
arAxisCtrl_gb[AxisNo.OutRobot_X].Admin._OpMode.en := ModeHoming;

//OutRobot Y

arAxisCtrl_gb[AxisNo.OutRobot_Y].Admin._OpMode.en := ModeHoming;

//RoundBelt

arAxisCtrl_gb[AxisNo.RoundBelt].Admin._OpMode.en := ModeHoming;

//TurnTable

arAxisCtrl_gb[AxisNo.TurnTable].Admin._OpMode.en := ModeHoming;
END_METHOD

METHOD ResetAction
VAR_OUTPUT
    xComplete : BOOL := TRUE;
END_VAR
AxisHomingRequest := FALSE;
uiCyclicStep := 0;
END_METHOD

METHOD StartAction
VAR_OUTPUT
    xComplete : BOOL := TRUE;
	iErrorID : INT := 0;
END_VAR
xComplete := FALSE;

uiCyclicStep := 0;
Homed := FALSE;

xComplete := TRUE;
END_METHOD

END_FUNCTION_BLOCK

// ---- Library/20_MachineUnits/22_AllocateArea/Service/FB_RoundBeltService.TcPOU
FUNCTION_BLOCK FB_RoundBeltService EXTENDS FB_ActionBasic
VAR_INPUT
    xExecute      : BOOL;
    xAbort        : BOOL;
    TargetStation : INT;

    Cylinder : REFERENCE TO UNI_CylinderList;
    TimeOut  : LREAL := 90; // Unit : s
	Pause	 : BOOL;
END_VAR
VAR_OUTPUT
    xAborted : BOOL;
    iErrorID : INT;
    ErrorMsg : STRING;
	AxisRoundMoveRequest	: BOOL;
END_VAR
VAR
    StateBehavior   : CBML.ETrigATo;
    CurrentPosition : ST_PositionTable;
    CurrentData     : ARRAY[1..21] OF ST_PositionTable;
    uiCyclicStep    : UINT := 0;
    uiIndexLoop     : UINT;
	fbExecuteEdgeDetect :FB_EdgeDetect;
	iVar	: INT;
	
	bWorkZonePlug_Extend	: BOOL;
	bWorkZonePress_Extend	: BOOL;
	bChargeZonePlug_Extend	: BOOL;
	
	TON_ServiceTimeOut		: TON;
	bServiceTimeOutIn		: BOOL;
END_VAR

THIS^.IBehaviourModel := StateBehavior;
StateBehavior(xExecute := xExecute,
              xAbort := xAbort OR fbExecuteEdgeDetect.xFallingEdge,
              udiTimeOut := LREAL_TO_UDINT( TimeOut*1000000),
              xDone => xDone,
              xBusy => xBusy,
              xError => xError,
              xAborted => xAborted);

//Make sure that C# turns off execute to shut down the service
fbExecuteEdgeDetect(xInput :=xExecute);

//Error Msg
iErrorID := StateBehavior._model.iErrorID;
ErrorMsg := M_GetErrorMsg(xErrorID := iErrorID);

			  
A00_ReadPositionData();

TON_ServiceTimeOut(IN:= bServiceTimeOutIn AND NOT Pause, PT := T#90S);

ACTION A00_ReadPositionData:
FOR uiIndexLoop := 1 TO 20 DO
    CurrentData[uiIndexLoop] := FUN_GetPositionTableData(PositionName := 'B', Index := UINT_TO_LREAL(uiIndexLoop), Clip := E_ClipNo.A);
END_FOR
END_ACTION

METHOD CleanupAction
VAR_INPUT
    xAbortProposed : BOOL;
    iErrorIDProposed: INT;
END_VAR
VAR_OUTPUT
    xComplete : BOOL := TRUE;
    xAbort: BOOL := xAbortProposed;
 	iErrorID : INT := iErrorIDProposed;
END_VAR
uiCyclicStep := 0;
END_METHOD

METHOD CyclicAction
VAR_INPUT
    itfTimingController : CBML.ITimingController;
END_VAR
VAR_OUTPUT
    xComplete : BOOL := TRUE;
    iErrorID : INT := 0;
END_VAR
xComplete := FALSE;

// 圓帶使用相關氣缸 安全卡控
IF bWorkZonePlug_Extend AND arAxisCtrl_gb[AxisNo.RoundBelt].Admin.Axis.Status.NotMoving THEN
	Cylinder.List.fbRoundBelt_WorkZone_Plug.M_Extend();
END_IF
IF bWorkZonePress_Extend AND arAxisCtrl_gb[AxisNo.RoundBelt].Admin.Axis.Status.NotMoving THEN
	Cylinder.List.fbRoundBelt_WorkZone_Press.M_Extend();
END_IF
IF bChargeZonePlug_Extend AND arAxisCtrl_gb[AxisNo.RoundBelt].Admin.Axis.Status.NotMoving THEN
	Cylinder.List.fbRoundBelt_ChargeZone_Plug.M_Extend();
END_IF

// Service Work Timer
bServiceTimeOutIn := TRUE;
IF TON_ServiceTimeOut.Q THEN
	iErrorID := GVL_ErrorCode.GC_ERR_TIMEOUT;
END_IF

CASE uiCyclicStep OF
	
    0:
		//Check if current station is same as target
		IF ABS(CurrentPosition.X_Pos -  arAxisCtrl_gb[AxisNo.RoundBelt].Admin.Axis.NcToPlc.ModuloSetPos) < 0.2 THEN
			uiCyclicStep := 200;
			ELSE
			uiCyclicStep := 50;	
		END_IF
	50:
		// Retract all cylinders
        Cylinder.List.fbRoundBelt_ChargeZone_Plug.M_Retract();
        Cylinder.List.fbRoundBelt_TransmitCVZone_Plug.M_Retract();
        Cylinder.List.fbRoundBelt_WorkZone_Plug.M_Retract();
        Cylinder.List.fbRoundBelt_WorkZone_Press.M_Retract();

        IF Cylinder.List.fbRoundBelt_ChargeZone_Plug.InRearPosition AND
            Cylinder.List.fbRoundBelt_TransmitCVZone_Plug.InRearPosition AND
            Cylinder.List.fbRoundBelt_WorkZone_Plug.InRearPosition AND
            Cylinder.List.fbRoundBelt_WorkZone_Press.InRearPosition THEN
            uiCyclicStep := 100;
        END_IF
    100: 
	    // Move round belt to target station
        arAxisCtrl_gb[AxisNo.RoundBelt].PosMode.Position := CurrentPosition.X_Pos;
		IF arAxisCtrl_gb[AxisNo.RoundBelt].PosMode.Position = CurrentPosition.X_Pos THEN
			uiCyclicStep := 125;
		END_IF
	125:
			AxisRoundMoveRequest := TRUE;
		 IF  arAxisCtrl_gb[AxisNo.RoundBelt].Admin.Axis.Status.Moving THEN
				uiCyclicStep := 150;
		 END_IF
		
	150:
        IF arAxisStatus_gb[AxisNo.RoundBelt].Admin._OpModeAck = ModePosAbs AND arAxisStatus_gb[AxisNo.RoundBelt].Admin.CmdDone AND
			(arAxisCtrl_gb[AxisNo.RoundBelt].Admin.Axis.Status.InTargetPosition OR arAxisCtrl_gb[AxisNo.RoundBelt].Admin.Axis.Status.Operational)
		THEN
			AxisRoundMoveRequest := FALSE;
            uiCyclicStep := 170;
        END_IF
		
	170:	// judge odd or even station

		IF iVar = 0 THEN
			uiCyclicStep := 400;
		ELSIF iVar = 1 THEN
			uiCyclicStep := 200;
		END_IF
		
	200:
        bChargeZonePlug_Extend 	:= TRUE;
		bWorkZonePlug_Extend	:= TRUE;
   
        IF Cylinder.List.fbRoundBelt_ChargeZone_Plug.InFrontPosition AND
            Cylinder.List.fbRoundBelt_WorkZone_Plug.InFrontPosition THEN
            uiCyclicStep := 300;
        END_IF
		
	300:
		bWorkZonePress_Extend	:= TRUE;
		
		IF  Cylinder.List.fbRoundBelt_WorkZone_Press.InFrontPosition THEN
			uiCyclicStep := 400;
        END_IF
	400:
			xComplete := TRUE;
			
			
END_CASE

IF arAxisCtrl_gb[AxisNo.RoundBelt].Admin.Axis.Status.Error THEN
    iErrorID := 6; // Axis RoundBelt has error
END_IF

IF Cylinder.List.fbRoundBelt_ChargeZone_Plug.xError THEN
    iErrorID := 7;
END_IF

IF Cylinder.List.fbRoundBelt_TransmitCVZone_Plug.xError THEN
    iErrorID := 8;
END_IF

IF Cylinder.List.fbRoundBelt_WorkZone_Plug.xError THEN
    iErrorID := 9;
END_IF

IF Cylinder.List.fbRoundBelt_WorkZone_Press.xError THEN
    iErrorID := 10;
END_IF
END_METHOD

METHOD ExitAction
VAR_INPUT
    xAfterCleanup : BOOL;
    xInCopyCode : BOOL;
END_VAR
END_METHOD

METHOD M_GetErrorMsg : T_MaxString
VAR_INPUT
	xErrorID: INT;
END_VAR

VAR
	
END_VAR
CASE xErrorID OF
	0:
		M_GetErrorMsg := 'No Error';
	1:
		M_GetErrorMsg := 'FB_RoundBeltService ErrorID 1: Action time out';
	2:
		M_GetErrorMsg := 'FB_RoundBeltService ErrorID 2: Position Data invalid';
	3:
		M_GetErrorMsg := 'FB_RoundBeltService ErrorID 3: Index invalid';
	4:
		M_GetErrorMsg := 'FB_RoundBeltService ErrorID 4: Axis roundbelt not ready has Error';
	5:
		M_GetErrorMsg := 'FB_RoundBeltService ErrorID 5: Cylinder not ready has Error';
	6:
		M_GetErrorMsg := 'FB_RoundBeltService ErrorID 6: Axis RoundBelt has Error';
	7:
		M_GetErrorMsg := 'FB_RoundBeltService ErrorID 7: ChargeZone_Plug has Error';
	8:
		M_GetErrorMsg := 'FB_RoundBeltService ErrorID 8: TransmitCVZone_Plug has Error';
	9:
		M_GetErrorMsg := 'FB_RoundBeltService ErrorID 9: WorkZone_Plug has Error';
	10:
		M_GetErrorMsg := 'FB_RoundBeltService ErrorID 10: WorkZone_Press has Error';
END_CASE
END_METHOD

METHOD PRIVATE M_StationModify : BOOL
VAR_INPUT
	TargetStation : INT;
END_VAR

VAR_OUTPUT
	ModifiedTargetStation : INT;
END_VAR
ModifiedTargetStation := (TargetStation/2)+1;
END_METHOD

METHOD ResetAction
VAR_OUTPUT
    xComplete : BOOL := TRUE;
END_VAR
bServiceTimeOutIn := false;
END_METHOD

METHOD StartAction
VAR_OUTPUT
    xComplete : BOOL := TRUE;
	iErrorID : INT := 0;
END_VAR

VAR
	ModifiedTargetPos : INT;
END_VAR
xComplete := FALSE;
M_StationModify(TargetStation,ModifiedTargetStation =>ModifiedTargetPos);

bWorkZonePlug_Extend 	:= FALSE;
bWorkZonePress_Extend	:= FALSE;
bChargeZonePlug_Extend	:= FALSE;
bServiceTimeOutIn 	   	:= false;

//verify C# Station command
iVar := TargetStation MOD 2 ;

IF TargetStation >= 1 AND TargetStation <= 40 THEN
    CurrentPosition := CurrentData[ModifiedTargetPos];
ELSE
    iErrorID := 3; // Target Station invalid.
    RETURN;
END_IF
uiCyclicStep := 0;

IF arAxisCtrl_gb[AxisNo.RoundBelt].Admin.Axis.Status.NotMoving AND
    NOT arAxisCtrl_gb[AxisNo.RoundBelt].Admin.Axis.Status.Error THEN
    xComplete := TRUE;
ELSE
    iErrorID := 4; // Axis not ready
END_IF

IF iVar = 0 THEN
	CurrentPosition.X_Pos := CurrentPosition.X_Pos + 65;
	xComplete := TRUE;
END_IF
IF iVar = 1 THEN
	CurrentPosition.X_Pos := CurrentPosition.X_Pos  ;
	xComplete := TRUE;
END_IF


//IF Cylinder.List.fbRoundBelt_ChargeZone_Plug.xBusy AND Cylinder.List.fbRoundBelt_TransmitCVZone_Plug.xBusy AND 
//	Cylinder.List.fbRoundBelt_WorkZone_Plug.xBusy AND Cylinder.List.fbRoundBelt_WorkZone_Press.xBusy AND NOT 
//	Cylinder.List.fbRoundBelt_ChargeZone_Plug.xError AND NOT Cylinder.List.fbRoundBelt_TransmitCVZone_Plug.xError
//	AND NOT Cylinder.List.fbRoundBelt_WorkZone_Plug.xError AND NOT Cylinder.List.fbRoundBelt_WorkZone_Press.xError THEN
//	iErrorID := 5; // Cylinder not ready
//END_IF
//xComplete := TRUE;
END_METHOD

END_FUNCTION_BLOCK

// ---- Library/20_MachineUnits/22_AllocateArea/Service/FB_TurnTableService.TcPOU
FUNCTION_BLOCK FB_TurnTableService EXTENDS FB_ActionBasic
VAR_INPUT
    xExecute      : BOOL;
    xAbort        : BOOL;
    iTurnTableTarget : INT;			//1=A ,2=B ,3=C ,4=D
	Pause		  : BOOL;
    Cylinder : REFERENCE TO UNI_CylinderList;
    //TimeOut  : LREAL := 30; // Unit : s
END_VAR
VAR_OUTPUT
    xAborted : BOOL;
    iErrorID : INT;
    ErrorMsg : STRING;
	bTurnTableMoveRequest	: BOOL;
END_VAR
VAR
    StateBehavior   : CBML.ETrigATo;
    CurrentPosition : ST_PositionTable;
	uiCyclicStep    : UINT := 0;
	PosCmd			: INT;
	
	bPress_Extend	: BOOL;
	
	TON_ServiceTimeOut		: TON;
	bServiceTimeOutIn		: BOOL;
	
	fNormAngle		: LREAL;	// 轉換過後的目標位置
	fCurrentAngle	: LREAL;	// 轉盤軸實際位置
	diTurns			: DINT;		// 計算轉盤軸走了多少圈數 >> 圈數
END_VAR

THIS^.IBehaviourModel := StateBehavior;
StateBehavior(xExecute := xExecute,
              xAbort := xAbort,
              udiTimeOut := (*LREAL_TO_UDINT( TimeOut*1000000)*),
              xDone => xDone,
              xBusy => xBusy,
              xError => xError,
              xAborted => xAborted);
			  
//Error Msg
iErrorID := StateBehavior._model.iErrorID;
ErrorMsg := M_GetErrorMsg(xErrorID := iErrorID);

TON_ServiceTimeOut(IN := bServiceTimeOutIn AND NOT Pause ,PT := T#30S);

METHOD CleanupAction
VAR_INPUT
    xAbortProposed : BOOL;
    iErrorIDProposed: INT;
END_VAR
VAR_OUTPUT
    xComplete : BOOL := TRUE;
    xAbort: BOOL := xAbortProposed;
 	iErrorID : INT := iErrorIDProposed;
END_VAR
bServiceTimeOutIn := false;
END_METHOD

METHOD CyclicAction
VAR_INPUT
    itfTimingController : CBML.ITimingController;
END_VAR
VAR_OUTPUT
    xComplete : BOOL := TRUE;
    iErrorID : INT := 0;
END_VAR
VAR_INST
	
END_VAR
xComplete := FALSE;

IF bPress_Extend 
AND arAxisCtrl_gb[AxisNo.RackMotor].Admin.Axis.Status.NotMoving 
AND NOT arAxisCtrl_gb[AxisNo.TurnTable].Admin.Axis.Status.Error THEN
	Cylinder.List.fbTurntable_Press.M_Extend();
END_IF

// Service Work Timer
bServiceTimeOutIn := TRUE;
IF TON_ServiceTimeOut.Q THEN
	iErrorID := GVL_ErrorCode.GC_ERR_TIMEOUT;
END_IF

CASE uiCyclicStep OF
    0:	// 轉盤氣缸init
		Cylinder.List.fbTurntable_Press.M_Retract();

        IF Cylinder.List.fbTurntable_Press.InRearPosition THEN
            uiCyclicStep := 100;
        END_IF
		
    100:	// 給轉盤軸位置
        arAxisCtrl_gb[AxisNo.TurnTable].PosMode.Position := PosCmd;
		uiCyclicStep := 125;
		
	125:	// 給轉盤軸運動命令，檢查是否有移動或者是否在同一站。
		bTurnTableMoveRequest := TRUE;
		
		diTurns := TRUNC(arAxisCtrl_gb[AxisNo.TurnTable].Admin.Axis.NcToPlc.ActPos / 360.0);
		fNormAngle := arAxisCtrl_gb[AxisNo.TurnTable].Admin.Axis.NcToPlc.ActPos - DINT_TO_LREAL(diTurns) * 360.0;
		
		IF fNormAngle < 0.0 THEN
			fNormAngle := fNormAngle + 360.0;
		END_IF
				
        IF arAxisCtrl_gb[AxisNo.TurnTable].Admin.Axis.Status.Moving  
			OR FUN_CheckInPos(ActPos  			:= fNormAngle,
							  TargetPos 		:= PosCmd,
							  ToleranceRange 	:= 0.1)
		THEN
            uiCyclicStep := 150;
        END_IF
		
	150:	//檢查是否完成移動
        IF arAxisStatus_gb[AxisNo.TurnTable].Admin._OpModeAck = ModePosAbs AND arAxisStatus_gb[AxisNo.TurnTable].Admin.CmdDone THEN
			bTurnTableMoveRequest := FALSE;
            uiCyclicStep := 200;
        END_IF
		
	200:	// 氣缸伸出
        bPress_Extend := TRUE;

        IF Cylinder.List.fbTurntable_Press.InFrontPosition THEN
            uiCyclicStep := 300;
        END_IF
		
	300:
			bPress_Extend := FALSE;
			xComplete 	  := TRUE;
END_CASE

IF arAxisCtrl_gb[AxisNo.TurnTable].Admin.Axis.Status.Error THEN
    iErrorID := 6; // Axis TurnTable has error
END_IF

//IF Cylinder.List.fbTurntable_Press.xError THEN
//    iErrorID := 7;	//Clinder Error
//END_IF
END_METHOD

METHOD ExitAction
VAR_INPUT
    xAfterCleanup : BOOL;
    xInCopyCode : BOOL;
END_VAR
bServiceTimeOutIn := false;
END_METHOD

METHOD M_GetErrorMsg : T_MaxString
VAR_INPUT
	xErrorID: INT;
END_VAR

VAR
	
END_VAR
CASE xErrorID OF
	0:
		M_GetErrorMsg := 'No Error';
	1:
		M_GetErrorMsg := 'FB_TurnTableService ErrorID 1: Action time out';
	2:
		M_GetErrorMsg := 'FB_TurnTableService ErrorID 2: Position Data invalid';
	3:
		M_GetErrorMsg := 'FB_TurnTableService ErrorID 3: TurnTableTarget invalid';
	4:
		M_GetErrorMsg := 'FB_TurnTableService ErrorID 4: Axis not ready';
	5:
		M_GetErrorMsg := 'FB_TurnTableService ErrorID 5: Cylinder not ready';
	6:
		M_GetErrorMsg := 'FB_TurnTableService ErrorID 6: Axis TurnTable has Error';
	7:
		M_GetErrorMsg := 'FB_TurnTableService ErrorID 7: fbTurntable_Press has Error';
END_CASE
END_METHOD

METHOD ResetAction
VAR_OUTPUT
    xComplete : BOOL := TRUE;
END_VAR
bServiceTimeOutIn := false;
END_METHOD

METHOD StartAction
VAR_OUTPUT
    xComplete : BOOL := TRUE;
	iErrorID : INT := 0;
END_VAR
xComplete := FALSE;

bPress_Extend		  := FALSE;
bTurnTableMoveRequest := FALSE;
bServiceTimeOutIn 	  := false;

IF NOT (iTurnTableTarget >= 1 AND iTurnTableTarget <= 4) THEN
    iErrorID := 3; // Target Station invalid.
    RETURN;
END_IF

IF NOT arAxisCtrl_gb[AxisNo.TurnTable].Admin.Axis.Status.NotMoving AND
     arAxisCtrl_gb[AxisNo.TurnTable].Admin.Axis.Status.Error THEN
    iErrorID := 4; // Axis not ready
END_IF

CASE iTurnTableTarget OF 
	1:	//A
		PosCmd :=0;
		xComplete := TRUE;
	2:	//B
		PosCmd :=270;
		xComplete := TRUE;
	3:	//C
		PosCmd :=180;
		xComplete := TRUE;
	4:	//D
		PosCmd :=90;
		xComplete := TRUE;
END_CASE


//IF Cylinder.List.fbTurntable_Press.xBusy AND  
//NOT Cylinder.List.fbTurntable_Press.xError  THEN
//	iErrorID := 5; // Cylinder not ready
//END_IF

uiCyclicStep := 0;
END_METHOD

END_FUNCTION_BLOCK

// ---- Library/99_Utilities/FUNCTION/FUN_CheckInPos.TcPOU
FUNCTION FUN_CheckInPos : Bool
VAR_INPUT
	ActPos : LREAL;
	TargetPos:LREAL;
	ToleranceRange : LREAL;
END_VAR
VAR
	MaxPos : LREAL;
	MinPos : LREAL;
END_VAR

MaxPos := TargetPos + ToleranceRange;
MinPos := TargetPos - ToleranceRange;
IF ActPos > MinPos AND ActPos < MaxPos THEN
	FUN_CheckInPos := TRUE;
ELSE
	FUN_CheckInPos := FALSE;
END_IF

END_FUNCTION

// ---- Library/20_MachineUnits/22_AllocateArea/Service/FB_AllocateMoveAutoBatchMode.TcPOU
FUNCTION_BLOCK FB_AllocateMoveAutoBatchMode EXTENDS FB_ObjectBase_V2
VAR_INPUT
//    Execute    :BOOL;   // True : This prog will start.
//    Abort      :BOOL;   // True : This prog will be abort.
//    Reset      :BOOL;   // True : This prog will be reset.
//    ObjectName :STRING; // Set this fb name(About it's action)
//	Pause				:BOOL;
	SimpleAllocateMode	:BOOL;
	bOccupied			: BOOL;	
	Clips 				: REFERENCE TO  ARRAY[0..3] OF FB_Cylinder;
	cylinders 			: REFERENCE TO  ARRAY[0..3] OF FB_Cylinder;
	//AllocateRobot :REFERENCE TO FB_xyRobot;
	//TurnTable : REFERENCE TO FB_RotateTable;
	//RoundBelt : REFERENCE TO FB_RoundBelt;
	TurnTable_Press		 		   : REFERENCE TO FB_Cylinder;
	RoundBelt_Press 			   : REFERENCE TO FB_Cylinder;
	AutoAllocateJobBatch_Ctrl      :st_AllocateMoveAutoBatchMode_Ctrl;
	INPUT            			   : REFERENCE TO ST_InputTable;
    OUTPUT           			   : REFERENCE TO ST_OutputTable;
	NrOfAllocateCylinder 		   : UINT :=4;
	CurrentData 				   : REFERENCE TO ST_SetupPara; // Componets setup parameter
	bAutoAllocateJobDryRun         : BOOL := FALSE;
	RoundBeltMoveJob_Status 		: ST_StatusBasic;
END_VAR

VAR_OUTPUT
//    Busy    :BOOL;        // True : This prog is running.
//    Done    :BOOL;        // True : Command has been executed.
//    Aborted :BOOL;        // True : This prog is aborted.
//    Error   :BOOL;        // True : This prog has an error.
//    ErrorID :UINT;       // Output ErrorID
//    Status  :T_MaxString; // Output this prog status by string(255bytes)
	RoundBeltMoveJob_Ctrl : ST_CommandBasic;
	RoundBeltMoveJob_Position	:LREAL;
	ProcessedIndex : ARRAY[0..49] OF INT;
	//UniqueErrorCode :STRING;
	// AutoAllocateJobBatch_Status    :st_AllocateMoveAutoBatchMode_Status;

END_VAR

VAR
//    eState :E_MethodStatus_Basic;
//	uiExecutingStep : UDINT; // This var is used to been controll STATE_EXECUTING process.
//	uiResettingStep : UDINT;
//	uiAbortingStep : UDINT;
//	_Executed :BOOL; // Executing process completed.
//	_Error : BOOL; // FB has an error.
//	_ResetCompleted : BOOL; // FB resetting completed.
//	_AbortCompleted : BOOL; // FB aborting completed.
//	_Abort		: BOOL;
	strStatus	: STRING;
	uiResumeStep : UINT;

//	bSimpleAllocationBatchEnable		 :BOOL;
//	AutoRotatebelt_Internal_Ctrl   : st_RoundBeltAutoSingleMove_Ctrl;
	_UniqueErrorCode : STRING;
	arrProcessedIndex : ARRAY[0..49] OF INT;
 //   eState              :E_MethodStatus_Basic;  
  //  uiAbortingStep      :UDINT;
    uiAbortedStep       :UDINT;
  //  uiResettingStep     :UDINT;
	uiResumableStep		: E_AllocationJob;
	_bRetry				: BOOL;
    bAborttingCompleted :BOOL; // True: Aborting process finished
    bAborted            :BOOL; // True : Aborted process finished
    bExecuted           :BOOL; // True : Executing process finished
    bResettingCompleted :BOOL; // True : Resetting process finished  
    iWorkingIndex		:UINT:=0;	
	iProcessingIndex	:INT :=0;
	iWorkingCylinder	:INT;
	//_Error				:BOOL :=FALSE;
	StatusDescription	:STRING;
	ClipsHaveNeedle		: ARRAY[0..3] OF BOOL;
	ClipsHaveNeedle_Pick		: ARRAY[0..3] OF BOOL;
	bCylinderCheck 		: BOOL;
	bCylinderCheckFastMode : BOOL;
	iPickingNeedleCount		:INT;
	iPlacingNeedleCount		:INT;
	bIfNextCycle			:BOOL;
	bCheckStation			:BOOL:=FALSE;
	
	
	tAutoAllocationJobBatchTimeOut :Tc2_Standard.TON;
    sAllocationJobBatchStatus      :STRING;
    tonFastModeTimeDelayBatch      :Tc2_Standard.TON;
	AllocationJobBatchMode		:E_AllocationJob := E_AllocationJob.Defult;
	 Ton_RoundBeltArrivedDelay     : TON;
	 CurrentPosition : ST_PositionTable;
	
  	RoundBeltMoveJob : st_AllocateCircleMoveStructure;	
	
		
//==========================M_AllocationJobBatchMode================================

	{attribute 'hide'}
	bCheckTrue : BOOL:=TRUE;
	iCurrentRotateBeltStation : UINT;
	i : UINT;	
	j : UINT;	

	bMoveRotateBeltBusy	:BOOL;
	bMoveRotateBeltDone : BOOL;
	A1Used				:BOOL :=FALSE;
	A2Used				:BOOL :=FALSE;
	R1Used				:BOOL :=FALSE;
	R2Used				:BOOL :=FALSE;
	bBoxCheck			:BOOL :=TRUE;
	PickingStation		:UINT;
	iNextPickingStation :UINT;
	
	

	
	
END_VAR

A00_BasicUnits();
SUPER^.A10_StateControl();

ACTION A00_BasicUnits:
Ton_RoundBeltArrivedDelay();
tonFastModeTimeDelayBatch();
tAutoAllocationJobBatchTimeOut(PT := T#60s);	//default 20s
END_ACTION

METHOD GetModelState
VAR_OUTPUT
    xDone    :BOOL;
    xBusy    :BOOL;
    xError   :BOOL;
    xAborted :BOOL;
    iErrorID :UDINT;
	UniqueErrorCode : STRING;
END_VAR
xDone    := Done;
xBusy    := Busy;
xError   := Error;
xAborted := Aborted;
iErrorID := ErrorID;
END_METHOD

METHOD GetName : STRING
GetName := ObjectName;
END_METHOD

(* Check Allocate Robot Clip cylinder no error
	Return True : no error
*)
METHOD M_CheckClipsNoError : BOOL
VAR_INPUT
END_VAR
//IF Clips[E_ClipsNo.ClipA].bError OR Clips[E_ClipsNo.ClipB].bError OR Clips[E_ClipsNo.ClipC].bError OR Clips[E_ClipsNo.ClipD].bError THEN
//    M_CheckClipsNoError := FALSE;
//ELSE
//    M_CheckClipsNoError := TRUE;
//END_IF
M_CheckClipsNoError := TRUE;
END_METHOD

(* Check Allocate Robot vertical cylinder no error
	return True : no error
*)
METHOD M_CheckCylindersNoError : BOOL
VAR_INPUT
END_VAR
//IF cylinders[E_CylinderNo.CylinderA].bError OR
//   cylinders[E_CylinderNo.CylinderB].bError OR
//   cylinders[E_CylinderNo.CylinderC].bError OR
//   cylinders[E_CylinderNo.CylinderD].bError
//THEN
//    M_CheckCylindersNoError := FALSE;
//ELSE
//    M_CheckCylindersNoError := TRUE;
//END_IF

M_CheckCylindersNoError := TRUE;
END_METHOD

METHOD PRIVATE M_RecoveryAxes : BOOL
VAR_INPUT
END_VAR
VAR
	bCheckTrue : BOOL;
	CheckErrorIndex : UINT;
END_VAR
bCheckTrue := TRUE;
FOR CheckErrorIndex:=1 TO 4 DO 
	IF arAxisCtrl_gb[CheckErrorIndex].Admin.Axis.Status.Error THEN
		arAxisCtrl_gb[CheckErrorIndex].Admin.ClearError:=TRUE;
		bCheckTrue:=FALSE;
	ELSE
		arAxisCtrl_gb[CheckErrorIndex].Admin.ClearError:=FALSE;	
	END_IF
END_FOR
//		TurnTable := 1,
//      RoundBelt := 2,
//      Allocate_X := 3,
//      Allocate_Y := 4,

M_RecoveryAxes:= bCheckTrue;
END_METHOD

METHOD  M_STATE_ABORTED
VAR_INPUT
END_VAR
IF NOT _bRetry THEN
	Busy     := FALSE;
	Aborted := TRUE;
	Status  := StatusDescription;
	Error   := TRUE;
	uiAbortingStep := 0;
	_AbortCompleted := FALSE;
END_IF

IF SimpleAllocateMode THEN
	ErrorID := 112;
ELSE
	ErrorID := 108;
END_IF

IF Reset THEN
	Aborted := FALSE;
	Error := FALSE;
	_bRetry := TRUE;
END_IF

IF NOT Execute THEN
	eState := STATE_RESETTING;
ELSIF Execute AND _bRetry THEN
	AllocationJobBatchMode := uiResumableStep;
	_bRetry := FALSE;
	eState := STATE_EXECUTING;
END_IF
END_METHOD

METHOD  M_STATE_ABORTING
VAR_INPUT
END_VAR
CASE uiAbortingStep OF
            0:
				_Abort := FALSE;
				_AbortCompleted := FALSE;
				_bRetry := FALSE;
				tAutoAllocationJobBatchTimeOut.IN:=FALSE;
				Ton_RoundBeltArrivedDelay.IN := FALSE;
				RoundBeltMoveJob.HandShake.Execute := FALSE;
				RoundBeltMoveJob_Ctrl.Execute := FALSE;
				
				uiAbortingStep:=100;
                // Aborting process start
                
			100:
//					FOR i:=1 TO GVL.NrOfAllocateCylinder DO
					
//					IF  clips[i].P_Error THEN clips[i].M_Reset('');	END_IF					
//					IF cylinders[i].P_Error THEN cylinders[i].M_Reset(''); END_IF
					
//				END_FOR
				FOR i:=0 TO 3 DO
					IF cylinders[i].xError THEN
						cylinders[i].M_Reset();
					ELSE
						cylinders[i].M_Retract();	
					END_IF
				END_FOR
					uiAbortingStep:=9000;
					
            9000:
                // Aborting process finished
                _AbortCompleted := TRUE;
        END_CASE

        IF NOT Execute THEN
            eState := STATE_RESETTING;
        ELSIF Execute AND _AbortCompleted THEN
            // Aborting process is running normally 
			uiAbortingStep:=0;
            eState := STATE_Aborted;
        ELSIF Error THEN
            // An error event occurred
            eState := STATE_ERROR;
        END_IF
END_METHOD

METHOD  M_STATE_DONE
VAR_INPUT
END_VAR
Busy := FALSE;
Done := TRUE;
RoundBeltMoveJob.HandShake.Execute:=FALSE;
RoundBeltMoveJob_Ctrl.Execute:= RoundBeltMoveJob.HandShake.Execute;
DAS_CoreSys.MachineControl.fbAllocateArea.M_ReleaseRoundBeltAccess(E_RoundBeltControlAccess.Allocating);
IF NOT Execute THEN
    eState := STATE_RESETTING;
END_IF
END_METHOD

METHOD  M_STATE_DORMANT
VAR_INPUT
END_VAR
VAR
	_arrProcessedIndex : ARRAY[0..49] OF INT;
END_VAR
Aborted         := FALSE;
Error           := FALSE;
ErrorID         := 0;
Busy                         := FALSE;
Done                         := FALSE;
_ResetCompleted := FALSE;
_Error          := FALSE;
_Executed       := FALSE;
_Abort			:= FALSE;
_AbortCompleted := FALSE;
_bRetry := FALSE;
Aborted			:= FALSE;
strStatus 		:='No Error';
Status          := '';

uiExecutingStep :=uiResettingStep :=uiResumeStep :=0;
AllocationJobBatchMode := E_AllocationJob.PreDataProcess;
i :=0;
j :=0;
iProcessingIndex :=0;
iWorkingCylinder :=0;
iWorkingIndex                := 0;	
Ton_RoundBeltArrivedDelay.IN := FALSE;
tAutoAllocationJobBatchTimeOut.IN := FALSE;

R1Used                       := FALSE;
R2Used                       := FALSE;
A1Used                       := FALSE;
A2Used                       := FALSE;
bMoveRotateBeltDone          := FALSE;	
bIfNextCycle				 := FALSE;	
bResettingCompleted :=false;
arrProcessedIndex :=_arrProcessedIndex;
IF Execute THEN
	
	eSTATE:=STATE_EXECUTING;
END_IF
END_METHOD

METHOD  M_STATE_ERROR
VAR_INPUT
END_VAR
VAR
	i : INT;
	RoundBelt_PressIF: INT;
END_VAR
Busy                         := FALSE;
Error                        := _Error;
tAutoAllocationJobBatchTimeOut.IN := FALSE;
Status                       := StatusDescription;
RoundBeltMoveJob.HandShake.Execute:=FALSE;
RoundBeltMoveJob_Ctrl.Execute:= RoundBeltMoveJob.HandShake.Execute;
DAS_CoreSys.MachineControl.fbAllocateArea.M_ReleaseRoundBeltAccess(E_RoundBeltControlAccess.Allocating);
FOR i:=0 TO 3 DO
	IF cylinders[i].xError THEN
		cylinders[i].M_Reset();
	ELSE
		cylinders[i].M_Retract();	
	END_IF
END_FOR

TurnTable_Press.M_Retract();
RoundBelt_Press.M_Retract();

IF NOT Execute THEN
    eState := STATE_RESETTING;
END_IF
END_METHOD

METHOD  M_STATE_EXECUTING
VAR_INPUT
END_VAR

VAR_INST	
	CurrentProcessData	: ST_AllocationJobBatchModeInfo;
	CurrentPickingCoordinates : ARRAY[0..3] OF st_Coordinate;
	CurrentPlacingCoordinates : ARRAY[0..3] OF st_Coordinate;
	CurrentSyncGroupPicking		  : ARRAY[0..3] OF UINT :=[0,1,2,3];
	CurrentSyncGroupPiacing		  : ARRAY[0..3] OF UINT :=[0,1,2,3];
END_VAR
		Busy := TRUE;

		// Pause gate:
		// 停止本 Service 繼續派發新動作,並關閉 timeout 計時。
		// 不清除圓帶的命令跟取消移動命令，以防暫停的不步序是在等待到位或者完成，避免卡死。
		IF Pause THEN
			Paused := TRUE;
			StatusDescription := 'Allocate batch reverse paused';
			tAutoAllocationJobBatchTimeOut.IN := FALSE;
			Ton_RoundBeltArrivedDelay.IN := FALSE;
//			RoundBeltMoveJob.HandShake.Execute := FALSE;
//			RoundBeltMoveJob_Ctrl.Execute := FALSE;
//			bAllocateRobotMoveRequest := FALSE;
			RETURN;
		END_IF
		Paused := FALSE;
			
		// 非自動模式直接中止 (避免軸控衝突)
		IF GVL_Machine.PackTags[UnitNo.Allocate].Status.UnitModeCurrent <> E_UnitMode.Auto THEN
			StatusDescription := 'FB_AllocateMoveAutoBatchMode, Not in Auto mode';
			_UniqueErrorCode := 'E_NOT_AUTO_MODE';
			_Error := TRUE;
		END_IF		
		
		tonFastModeTimeDelayBatch.PT:=T#10MS;
		ProcessedIndex:=arrProcessedIndex;
		IF NOT bAutoAllocateJobDryRun THEN
			DAS_CoreSys.MachineControl.fbAllocateArea.M_GetRoundBeltAccess(E_RoundBeltControlAccess.Allocating);	
			RoundBeltMoveJob_Position:= RoundBeltMoveJob.Position;
			RoundBeltMoveJob_Ctrl.Execute:= RoundBeltMoveJob.HandShake.Execute;
			RoundBeltMoveJob_Ctrl.Reset:= RoundBeltMoveJob.HandShake.Reset;	
			RoundBeltMoveJob.HandShake.Busy :=RoundBeltMoveJob_Status.Busy;
			RoundBeltMoveJob.HandShake.Done :=RoundBeltMoveJob_Status.Done;
			RoundBeltMoveJob.HandShake.Error :=RoundBeltMoveJob_Status.Error;	
	
		END_IF
		
		CASE AllocationJobBatchMode OF
			
			E_AllocationJob.PreDataProcess:			
			
				IF NOT Pause THEN // Pausing here waiting pause finish
					
					bCheckStation:=FALSE;
					//Get current allocation data
					FOR i:=iProcessingIndex TO AutoAllocateJobBatch_Ctrl.AutoMode_AllocateMoveBatch.NrOfAllocationJob-1 BY 1  DO
						CurrentProcessData :=AutoAllocateJobBatch_Ctrl.AutoMode_AllocateMoveBatch.AllocationInfo[iProcessingIndex];
						
						FOR j:=0 TO 3 DO
							IF NOT (CurrentProcessData.PickingNeedleInfo[j].Station=99) THEN
									bCheckStation:=TRUE; //Station = 99 means this job should be ignou , Therefor any station of job is "not" 99 , means this job should be process
								EXIT;
							END_IF						
						END_FOR
						
						IF bCheckStation THEN // CheckStation = true means this job is vaild 
								AllocationJobBatchMode:=E_AllocationJob.Idle;
								EXIT;
							ELSE // Other wise , this job is no need to process , just go check next job
								iProcessingIndex:=iProcessingIndex+1;
								arrProcessedIndex[i] :=CurrentProcessData.ID;
						END_IF						
					END_FOR		

					IF 	AutoAllocateJobBatch_Ctrl.AutoMode_AllocateMoveBatch.NrOfAllocationJob<= iProcessingIndex THEN
							AllocationJobBatchMode:=E_AllocationJob.Finish; // If all jobs was processed or checked , Batch jobs done
					END_IF				
				END_IF
				
			E_AllocationJob.Idle:
				//idle 
				FOR i :=0 TO 3 DO
						
						FUN_GetNeedleCoordinates(uiLocation:=0,	// Location 0 : Rotate belt , 1 : turn table
										uiBox:=CurrentProcessData.PickingNeedleInfo[i].Box,
										uiClip:=CurrentProcessData.PickingNeedleInfo[i].Clip,
										uiNeedleLocation :=CurrentProcessData.PickingNeedleInfo[i].NeedleLocation,
										NeedleCoordinate=>CurrentPickingCoordinates[i]);
						// Get picking coordinate , always from rotate belt
				
						IF SimpleAllocateMode THEN // Get placing coordinate , if working mode Simple allocate : Place to rotate belt
								FUN_GetNeedleCoordinates(uiLocation:=0,
										uiBox:=CurrentProcessData.PlacingNeedleInfo[i].Box,
										uiClip:=CurrentProcessData.PlacingNeedleInfo[i].Clip,
										uiNeedleLocation :=CurrentProcessData.PlacingNeedleInfo[i].NeedleLocation,
										NeedleCoordinate=>CurrentPlacingCoordinates[i]);
						ELSE	//Otherwias , place to turn table
								FUN_GetNeedleCoordinates(uiLocation:=1,
										uiBox:=CurrentProcessData.PlacingNeedleInfo[i].Box,
										uiClip:=CurrentProcessData.PlacingNeedleInfo[i].Clip,
										uiNeedleLocation :=CurrentProcessData.PlacingNeedleInfo[i].NeedleLocation,
										NeedleCoordinate=>CurrentPlacingCoordinates[i]);
						END_IF
										
									
